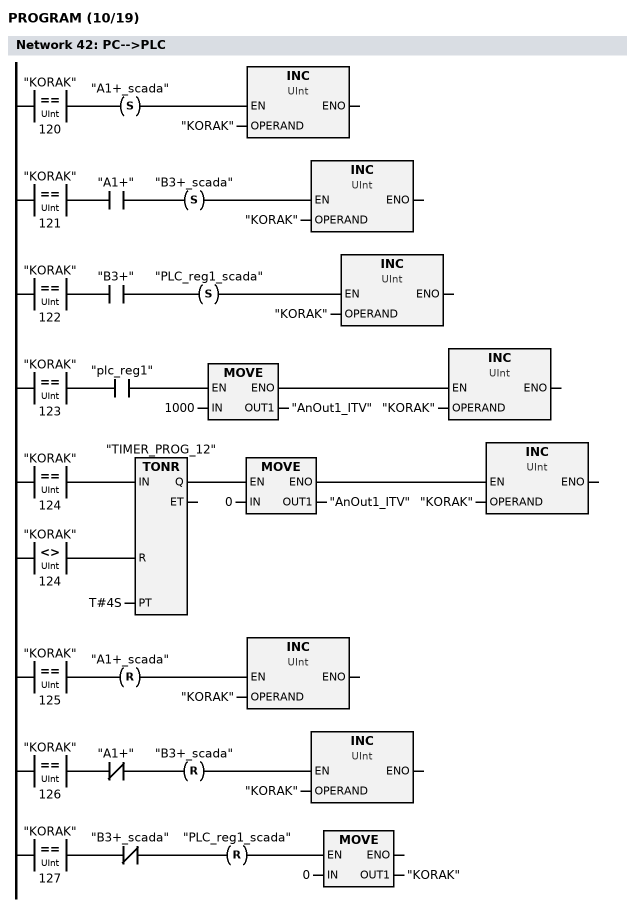
   IF "KORAK" = 120 THEN
       "A1+_scada" := TRUE;
       "KORAK" := "KORAK" + 1;
   END_IF;
   IF ("KORAK" = 121) AND "A1+" THEN
       "B3+_scada" := TRUE;
       "KORAK" := "KORAK" + 1;
   END_IF;
   IF ("KORAK" = 122) AND "B3+" THEN
       "PLC_reg1_scada" := TRUE;
       "KORAK" := "KORAK" + 1;
   END_IF;
   IF ("KORAK" = 123) AND "plc_reg1" THEN
       "AnOut1_ITV" := 1000;
       "KORAK" := "KORAK" + 1;
   END_IF;
   "TIMER_PROG_12".TONR(IN := "KORAK" = 124, R := "KORAK" <> 124, PT := T#4S);
   IF "TIMER_PROG_12".Q THEN
       "AnOut1_ITV" := 0;
       "KORAK" := "KORAK" + 1;
   END_IF;
   IF "KORAK" = 125 THEN
       "A1+_scada" := FALSE;
       "KORAK" := "KORAK" + 1;
   END_IF;
   IF ("KORAK" = 126) AND NOT "A1+" THEN
       "B3+_scada" := FALSE;
       "KORAK" := "KORAK" + 1;
   END_IF;
   IF ("KORAK" = 127) AND NOT "B3+_scada" THEN
       "PLC_reg1_scada" := FALSE;
       "KORAK" := 0;
   END_IF;
END_REGION

REGION Network 43: PC-->PLC
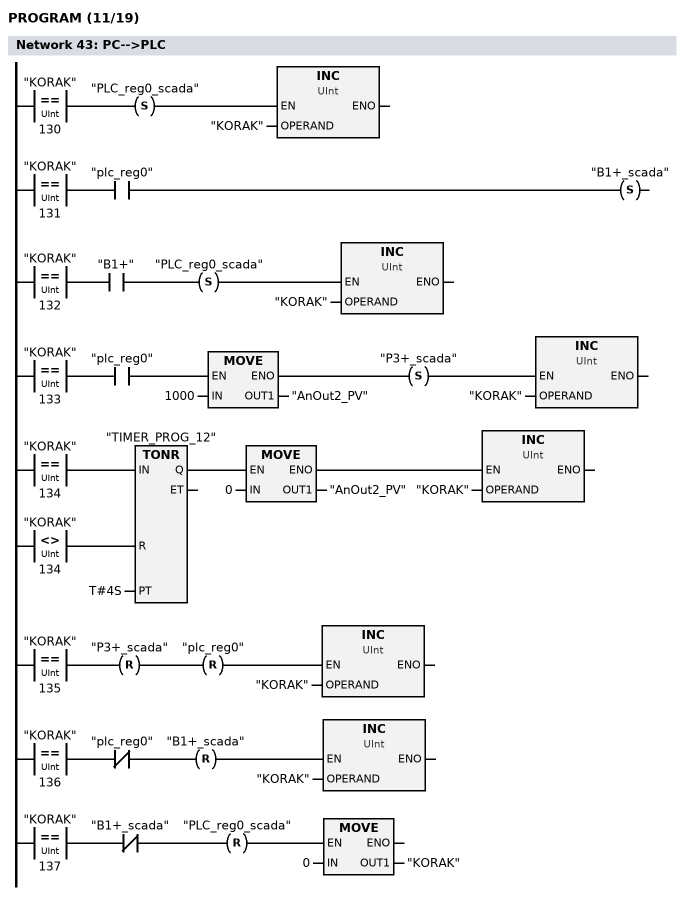
   IF "KORAK" = 130 THEN
       "PLC_reg0_scada" := TRUE;
       "KORAK" := "KORAK" + 1;
   END_IF;
   IF ("KORAK" = 131) AND "plc_reg0" THEN "B1+_scada" := TRUE; END_IF;
   IF ("KORAK" = 132) AND "B1+" THEN
       "PLC_reg0_scada" := TRUE;
       "KORAK" := "KORAK" + 1;
   END_IF;
   IF ("KORAK" = 133) AND "plc_reg0" THEN
       "AnOut2_PV" := 1000;
       "P3+_scada" := TRUE;
       "KORAK" := "KORAK" + 1;
   END_IF;
   "TIMER_PROG_12".TONR(IN := "KORAK" = 134, R := "KORAK" <> 134, PT := T#4S);
   IF "TIMER_PROG_12".Q THEN
       "AnOut2_PV" := 0;
       "KORAK" := "KORAK" + 1;
   END_IF;
   IF "KORAK" = 135 THEN
       "P3+_scada" := FALSE;
       "plc_reg0" := FALSE;
       "KORAK" := "KORAK" + 1;
   END_IF;
   IF ("KORAK" = 136) AND NOT "plc_reg0" THEN
       "B1+_scada" := FALSE;
       "KORAK" := "KORAK" + 1;
   END_IF;
   IF ("KORAK" = 137) AND NOT "B1+_scada" THEN
       "PLC_reg0_scada" := FALSE;
       "KORAK" := 0;
   END_IF;
END_REGION

REGION Network 44: PC-->PLC
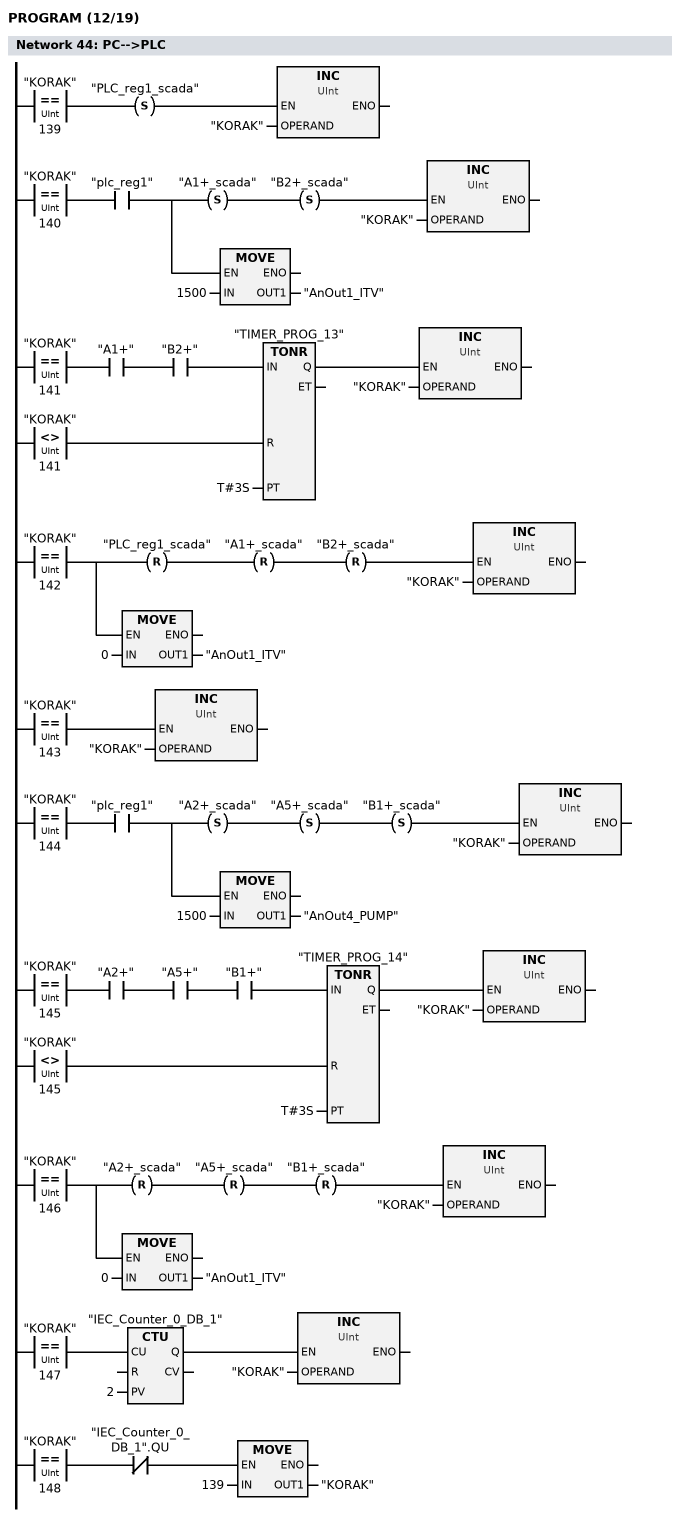
   IF "KORAK" = 139 THEN
       "PLC_reg1_scada" := TRUE;
       "KORAK" := "KORAK" + 1;
   END_IF;
   IF ("KORAK" = 140) AND "plc_reg1" THEN
       "A1+_scada" := TRUE;
       "B2+_scada" := TRUE;
   END_IF;
   #_w1 := ("KORAK" = 140) AND "plc_reg1";
   IF #_w1 THEN
       "KORAK" := "KORAK" + 1;
       "AnOut1_ITV" := 1500;
   END_IF;
   "TIMER_PROG_13".TONR(IN := ("KORAK" = 141) AND "A1+" AND "B2+", R := "KORAK" <> 141, PT := T#3S);
   IF "TIMER_PROG_13".Q THEN "KORAK" := "KORAK" + 1; END_IF;
   IF "KORAK" = 142 THEN
       "PLC_reg1_scada" := FALSE;
       "A1+_scada" := FALSE;
       "B2+_scada" := FALSE;
   END_IF;
   #_w2 := "KORAK" = 142;
   IF #_w2 THEN
       "KORAK" := "KORAK" + 1;
       "AnOut1_ITV" := 0;
   END_IF;
   IF "KORAK" = 143 THEN "KORAK" := "KORAK" + 1; END_IF;
   IF ("KORAK" = 144) AND "plc_reg1" THEN
       "A2+_scada" := TRUE;
       "A5+_scada" := TRUE;
       "B1+_scada" := TRUE;
   END_IF;
   #_w3 := ("KORAK" = 144) AND "plc_reg1";
   IF #_w3 THEN
       "KORAK" := "KORAK" + 1;
       "AnOut4_PUMP" := 1500;
   END_IF;
   "TIMER_PROG_14".TONR(IN := ("KORAK" = 145) AND "A2+" AND "A5+" AND "B1+", R := "KORAK" <> 145, PT := T#3S);
   IF "TIMER_PROG_14".Q THEN "KORAK" := "KORAK" + 1; END_IF;
   IF "KORAK" = 146 THEN
       "A2+_scada" := FALSE;
       "A5+_scada" := FALSE;
       "B1+_scada" := FALSE;
   END_IF;
   #_w4 := "KORAK" = 146;
   IF #_w4 THEN
       "KORAK" := "KORAK" + 1;
       "AnOut1_ITV" := 0;
   END_IF;
   "IEC_Counter_0_DB_1".CTU(CU := "KORAK" = 147, PV := 2);
   IF "IEC_Counter_0_DB_1".Q THEN "KORAK" := "KORAK" + 1; END_IF;
   IF ("KORAK" = 148) AND NOT "IEC_Counter_0_DB_1".QU THEN "KORAK" := 139; END_IF;
END_REGION

REGION Network 45: 2024_prva grupa
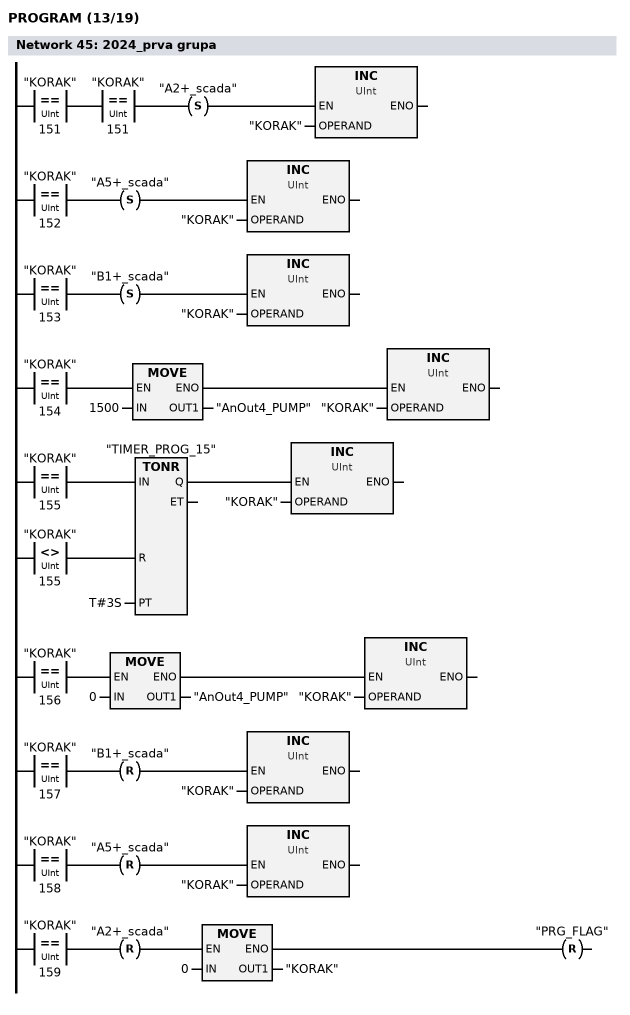
   IF ("KORAK" = 151) AND ("KORAK" = 151) THEN
       "A2+_scada" := TRUE;
       "KORAK" := "KORAK" + 1;
   END_IF;
   IF "KORAK" = 152 THEN
       "A5+_scada" := TRUE;
       "KORAK" := "KORAK" + 1;
   END_IF;
   IF "KORAK" = 153 THEN
       "B1+_scada" := TRUE;
       "KORAK" := "KORAK" + 1;
   END_IF;
   IF "KORAK" = 154 THEN
       "AnOut4_PUMP" := 1500;
       "KORAK" := "KORAK" + 1;
   END_IF;
   "TIMER_PROG_15".TONR(IN := "KORAK" = 155, R := "KORAK" <> 155, PT := T#3S);
   IF "TIMER_PROG_15".Q THEN "KORAK" := "KORAK" + 1; END_IF;
   IF "KORAK" = 156 THEN
       "AnOut4_PUMP" := 0;
       "KORAK" := "KORAK" + 1;
   END_IF;
   IF "KORAK" = 157 THEN
       "B1+_scada" := FALSE;
       "KORAK" := "KORAK" + 1;
   END_IF;
   IF "KORAK" = 158 THEN
       "A5+_scada" := FALSE;
       "KORAK" := "KORAK" + 1;
   END_IF;
   IF "KORAK" = 159 THEN "A2+_scada" := FALSE; END_IF;
   #_w1 := "KORAK" = 159;
   IF #_w1 THEN
       "KORAK" := 0;
       "PRG_FLAG" := FALSE;
   END_IF;
END_REGION

REGION Network 46: PC-->PLC
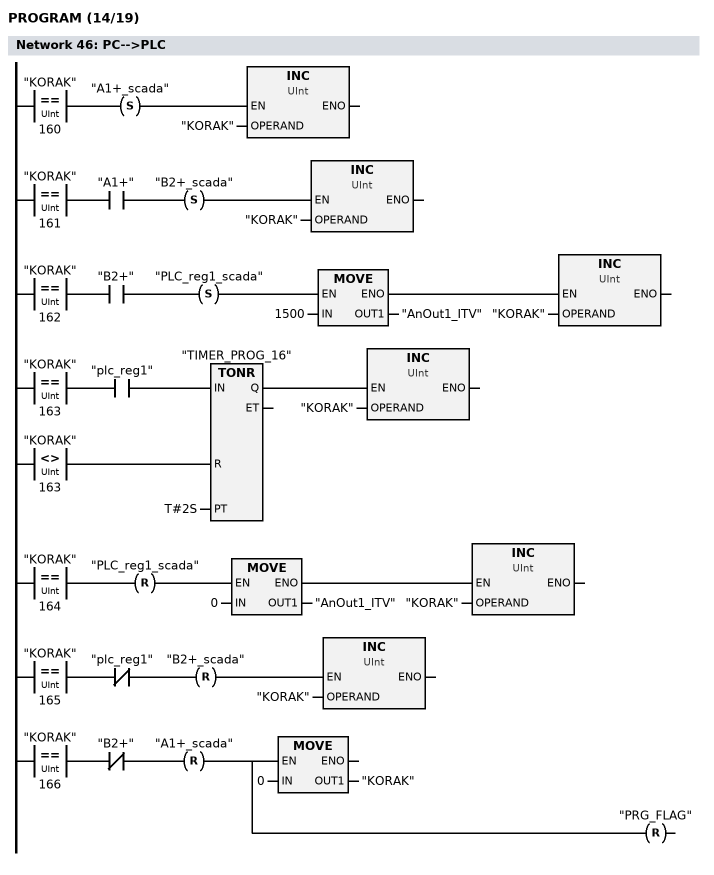
   IF "KORAK" = 160 THEN
       "A1+_scada" := TRUE;
       "KORAK" := "KORAK" + 1;
   END_IF;
   IF ("KORAK" = 161) AND "A1+" THEN
       "B2+_scada" := TRUE;
       "KORAK" := "KORAK" + 1;
   END_IF;
   IF ("KORAK" = 162) AND "B2+" THEN
       "PLC_reg1_scada" := TRUE;
       "AnOut1_ITV" := 1500;
       "KORAK" := "KORAK" + 1;
   END_IF;
   "TIMER_PROG_16".TONR(IN := ("KORAK" = 163) AND "plc_reg1", R := "KORAK" <> 163, PT := T#2S);
   IF "TIMER_PROG_16".Q THEN "KORAK" := "KORAK" + 1; END_IF;
   IF "KORAK" = 164 THEN
       "PLC_reg1_scada" := FALSE;
       "AnOut1_ITV" := 0;
       "KORAK" := "KORAK" + 1;
   END_IF;
   IF ("KORAK" = 165) AND NOT "plc_reg1" THEN
       "B2+_scada" := FALSE;
       "KORAK" := "KORAK" + 1;
   END_IF;
   IF ("KORAK" = 166) AND NOT "B2+" THEN "A1+_scada" := FALSE; END_IF;
   #_w1 := ("KORAK" = 166) AND NOT "B2+";
   IF #_w1 THEN
       "KORAK" := 0;
       "PRG_FLAG" := FALSE;
   END_IF;
END_REGION

REGION Network 47: PC-->PLC
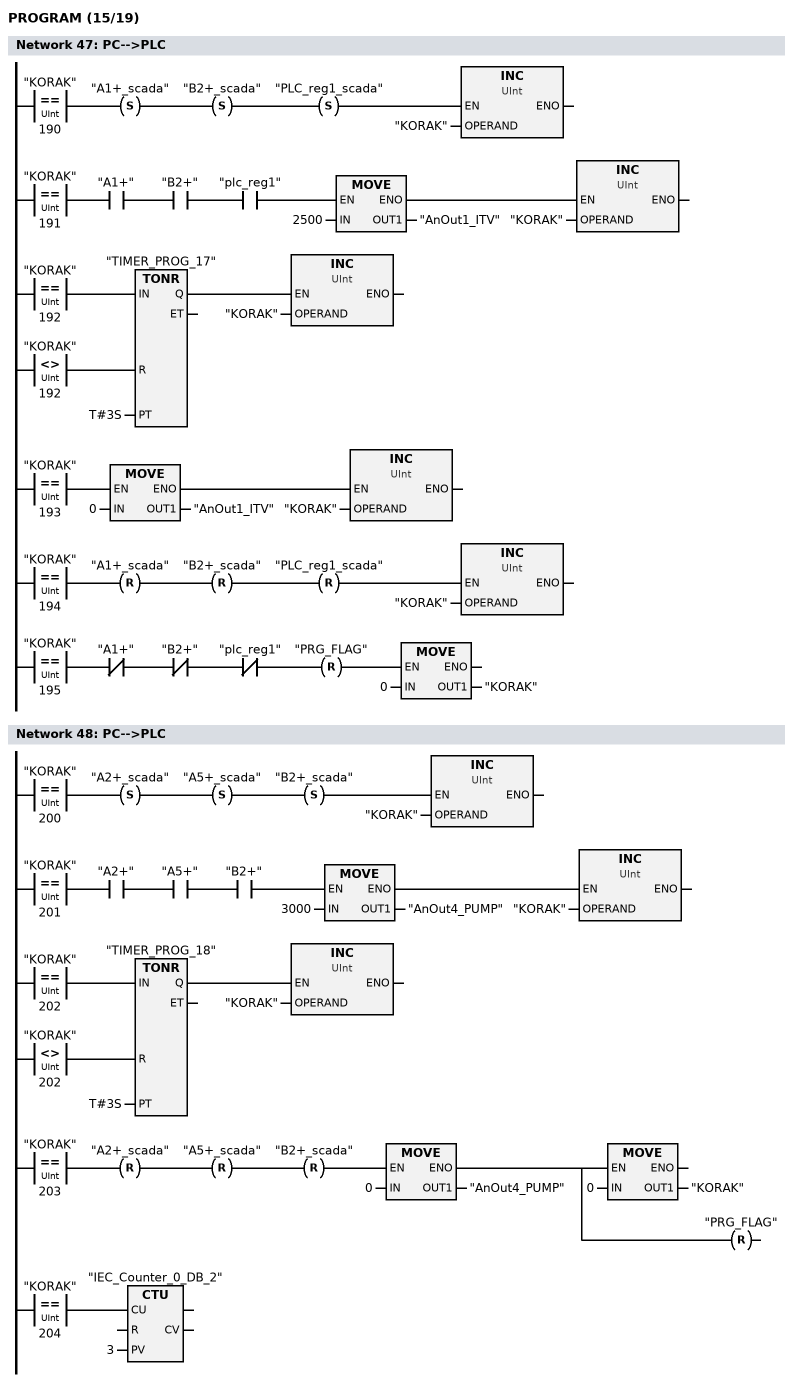
   IF "KORAK" = 190 THEN
       "A1+_scada" := TRUE;
       "B2+_scada" := TRUE;
       "PLC_reg1_scada" := TRUE;
       "KORAK" := "KORAK" + 1;
   END_IF;
   IF ("KORAK" = 191) AND "A1+" AND "B2+" AND "plc_reg1" THEN
       "AnOut1_ITV" := 2500;
       "KORAK" := "KORAK" + 1;
   END_IF;
   "TIMER_PROG_17".TONR(IN := "KORAK" = 192, R := "KORAK" <> 192, PT := T#3S);
   IF "TIMER_PROG_17".Q THEN "KORAK" := "KORAK" + 1; END_IF;
   IF "KORAK" = 193 THEN
       "AnOut1_ITV" := 0;
       "KORAK" := "KORAK" + 1;
   END_IF;
   IF "KORAK" = 194 THEN
       "A1+_scada" := FALSE;
       "B2+_scada" := FALSE;
       "PLC_reg1_scada" := FALSE;
       "KORAK" := "KORAK" + 1;
   END_IF;
   IF ("KORAK" = 195) AND NOT "A1+" AND NOT "B2+" AND NOT "plc_reg1" THEN
       "PRG_FLAG" := FALSE;
       "KORAK" := 0;
   END_IF;
END_REGION

REGION Network 48: PC-->PLC
   IF "KORAK" = 200 THEN
       "A2+_scada" := TRUE;
       "A5+_scada" := TRUE;
       "B2+_scada" := TRUE;
       "KORAK" := "KORAK" + 1;
   END_IF;
   IF ("KORAK" = 201) AND "A2+" AND "A5+" AND "B2+" THEN
       "AnOut4_PUMP" := 3000;
       "KORAK" := "KORAK" + 1;
   END_IF;
   "TIMER_PROG_18".TONR(IN := "KORAK" = 202, R := "KORAK" <> 202, PT := T#3S);
   IF "TIMER_PROG_18".Q THEN "KORAK" := "KORAK" + 1; END_IF;
   IF "KORAK" = 203 THEN
       "A2+_scada" := FALSE;
       "A5+_scada" := FALSE;
       "B2+_scada" := FALSE;
       "AnOut4_PUMP" := 0;
   END_IF;
   #_w1 := "KORAK" = 203;
   IF #_w1 THEN
       "KORAK" := 0;
       "PRG_FLAG" := FALSE;
   END_IF;
   "IEC_Counter_0_DB_2".CTU(CU := "KORAK" = 204, PV := 3);
END_REGION

REGION Network 49: PC-->PLC
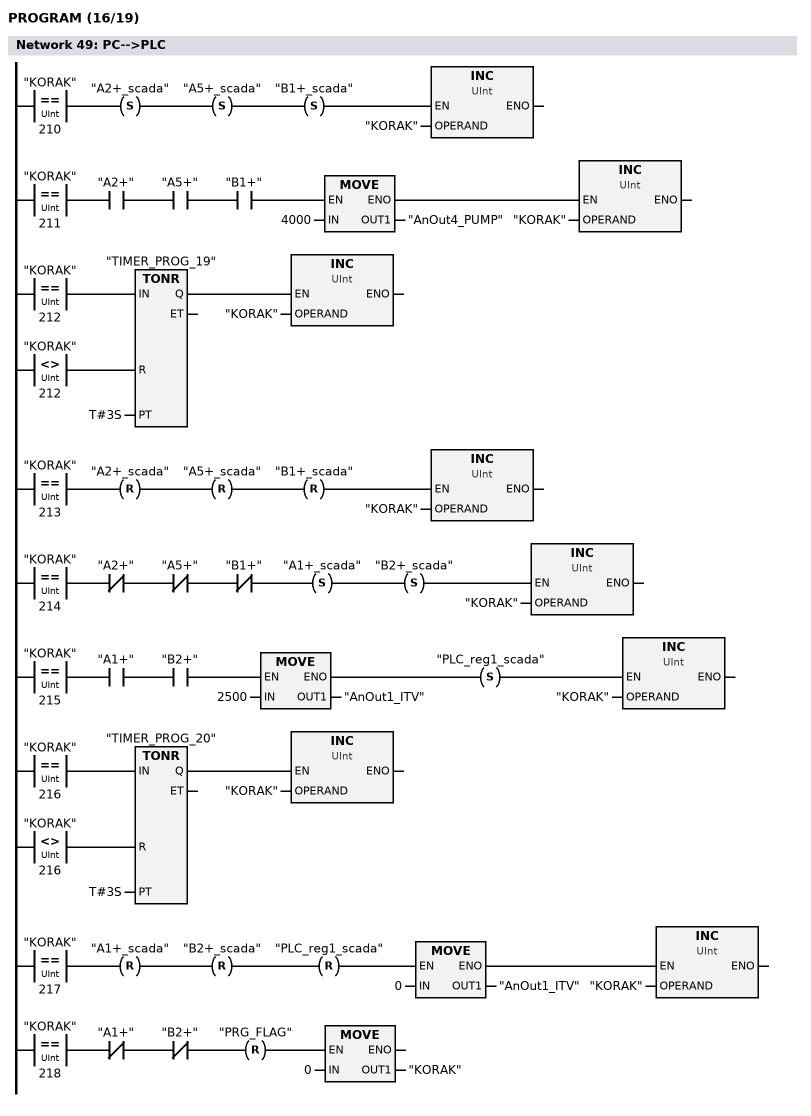
   IF "KORAK" = 210 THEN
       "A2+_scada" := TRUE;
       "A5+_scada" := TRUE;
       "B1+_scada" := TRUE;
       "KORAK" := "KORAK" + 1;
   END_IF;
   IF ("KORAK" = 211) AND "A2+" AND "A5+" AND "B1+" THEN
       "AnOut4_PUMP" := 4000;
       "KORAK" := "KORAK" + 1;
   END_IF;
   "TIMER_PROG_19".TONR(IN := "KORAK" = 212, R := "KORAK" <> 212, PT := T#3S);
   IF "TIMER_PROG_19".Q THEN "KORAK" := "KORAK" + 1; END_IF;
   IF "KORAK" = 213 THEN
       "A2+_scada" := FALSE;
       "A5+_scada" := FALSE;
       "B1+_scada" := FALSE;
       "KORAK" := "KORAK" + 1;
   END_IF;
   IF ("KORAK" = 214) AND NOT "A2+" AND NOT "A5+" AND NOT "B1+" THEN
       "A1+_scada" := TRUE;
       "B2+_scada" := TRUE;
       "KORAK" := "KORAK" + 1;
   END_IF;
   IF ("KORAK" = 215) AND "A1+" AND "B2+" THEN
       "AnOut1_ITV" := 2500;
       "PLC_reg1_scada" := TRUE;
       "KORAK" := "KORAK" + 1;
   END_IF;
   "TIMER_PROG_20".TONR(IN := "KORAK" = 216, R := "KORAK" <> 216, PT := T#3S);
   IF "TIMER_PROG_20".Q THEN "KORAK" := "KORAK" + 1; END_IF;
   IF "KORAK" = 217 THEN
       "A1+_scada" := FALSE;
       "B2+_scada" := FALSE;
       "PLC_reg1_scada" := FALSE;
       "AnOut1_ITV" := 0;
       "KORAK" := "KORAK" + 1;
   END_IF;
   IF ("KORAK" = 218) AND NOT "A1+" AND NOT "B2+" THEN
       "PRG_FLAG" := FALSE;
       "KORAK" := 0;
   END_IF;
END_REGION

REGION Network 50: PC-->PLC
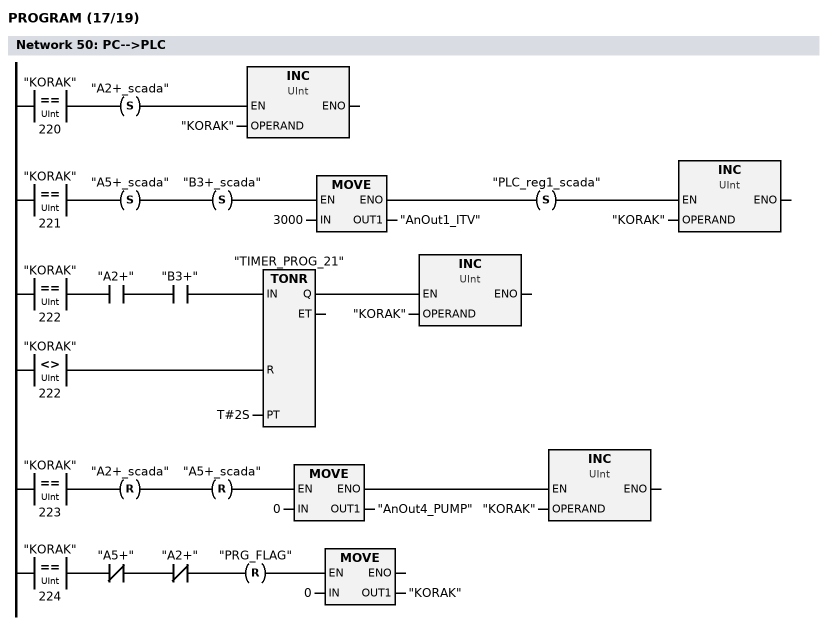
   IF "KORAK" = 220 THEN
       "A2+_scada" := TRUE;
       "KORAK" := "KORAK" + 1;
   END_IF;
   IF "KORAK" = 221 THEN
       "A5+_scada" := TRUE;
       "B3+_scada" := TRUE;
       "AnOut1_ITV" := 3000;
       "PLC_reg1_scada" := TRUE;
       "KORAK" := "KORAK" + 1;
   END_IF;
   "TIMER_PROG_21".TONR(IN := ("KORAK" = 222) AND "A2+" AND "B3+", R := "KORAK" <> 222, PT := T#2S);
   IF "TIMER_PROG_21".Q THEN "KORAK" := "KORAK" + 1; END_IF;
   IF "KORAK" = 223 THEN
       "A2+_scada" := FALSE;
       "A5+_scada" := FALSE;
       "AnOut4_PUMP" := 0;
       "KORAK" := "KORAK" + 1;
   END_IF;
   IF ("KORAK" = 224) AND NOT "A5+" AND NOT "A2+" THEN
       "PRG_FLAG" := FALSE;
       "KORAK" := 0;
   END_IF;
END_REGION

REGION Network 51: PC-->PLC
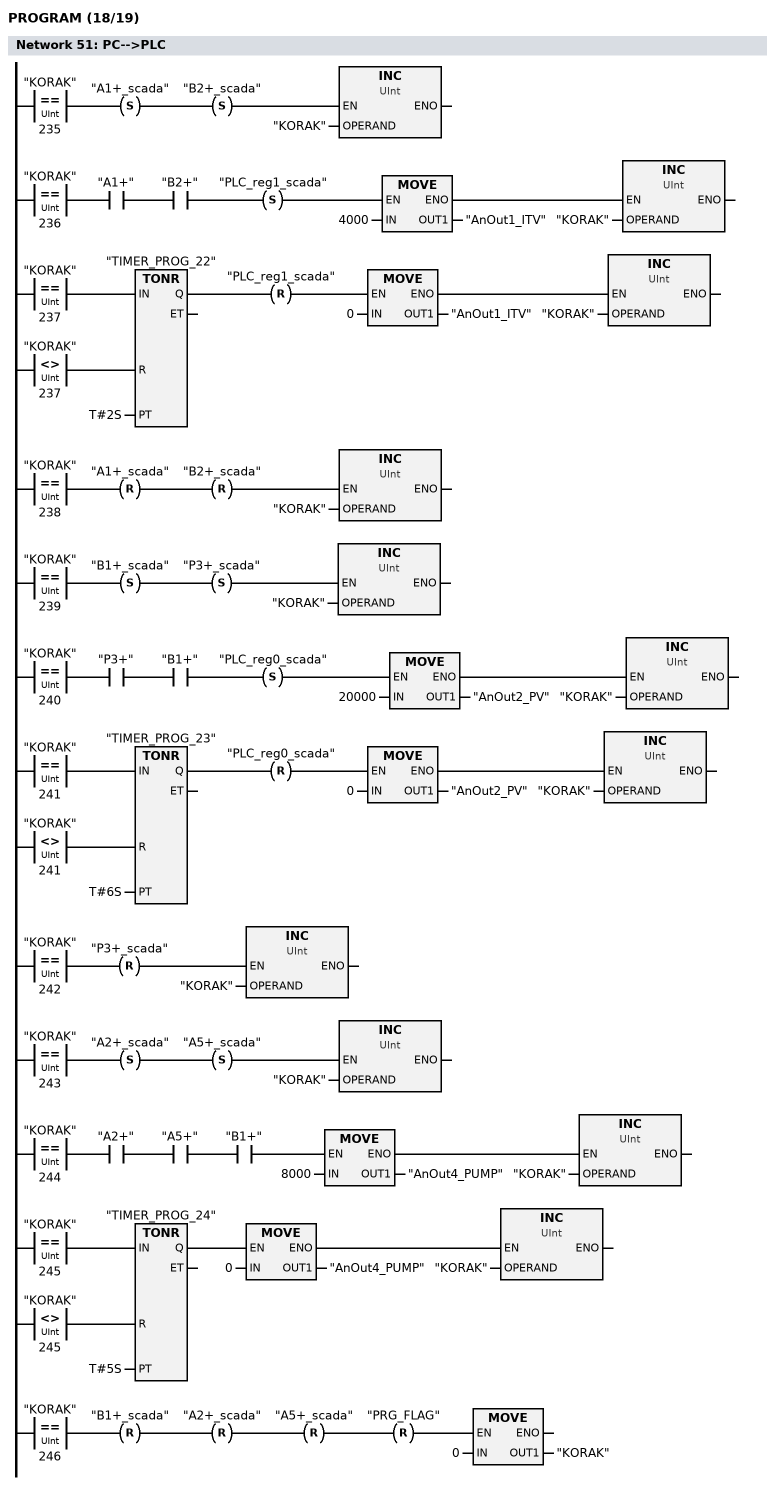
   IF "KORAK" = 235 THEN
       "A1+_scada" := TRUE;
       "B2+_scada" := TRUE;
       "KORAK" := "KORAK" + 1;
   END_IF;
   IF ("KORAK" = 236) AND "A1+" AND "B2+" THEN
       "PLC_reg1_scada" := TRUE;
       "AnOut1_ITV" := 4000;
       "KORAK" := "KORAK" + 1;
   END_IF;
   "TIMER_PROG_22".TONR(IN := "KORAK" = 237, R := "KORAK" <> 237, PT := T#2S);
   IF "TIMER_PROG_22".Q THEN
       "PLC_reg1_scada" := FALSE;
       "AnOut1_ITV" := 0;
       "KORAK" := "KORAK" + 1;
   END_IF;
   IF "KORAK" = 238 THEN
       "A1+_scada" := FALSE;
       "B2+_scada" := FALSE;
       "KORAK" := "KORAK" + 1;
   END_IF;
   IF "KORAK" = 239 THEN
       "B1+_scada" := TRUE;
       "P3+_scada" := TRUE;
       "KORAK" := "KORAK" + 1;
   END_IF;
   IF ("KORAK" = 240) AND "P3+" AND "B1+" THEN
       "PLC_reg0_scada" := TRUE;
       "AnOut2_PV" := 20000;
       "KORAK" := "KORAK" + 1;
   END_IF;
   "TIMER_PROG_23".TONR(IN := "KORAK" = 241, R := "KORAK" <> 241, PT := T#6S);
   IF "TIMER_PROG_23".Q THEN
       "PLC_reg0_scada" := FALSE;
       "AnOut2_PV" := 0;
       "KORAK" := "KORAK" + 1;
   END_IF;
   IF "KORAK" = 242 THEN
       "P3+_scada" := FALSE;
       "KORAK" := "KORAK" + 1;
   END_IF;
   IF "KORAK" = 243 THEN
       "A2+_scada" := TRUE;
       "A5+_scada" := TRUE;
       "KORAK" := "KORAK" + 1;
   END_IF;
   IF ("KORAK" = 244) AND "A2+" AND "A5+" AND "B1+" THEN
       "AnOut4_PUMP" := 8000;
       "KORAK" := "KORAK" + 1;
   END_IF;
   "TIMER_PROG_24".TONR(IN := "KORAK" = 245, R := "KORAK" <> 245, PT := T#5S);
   IF "TIMER_PROG_24".Q THEN
       "AnOut4_PUMP" := 0;
       "KORAK" := "KORAK" + 1;
   END_IF;
   IF "KORAK" = 246 THEN
       "B1+_scada" := FALSE;
       "A2+_scada" := FALSE;
       "A5+_scada" := FALSE;
       "PRG_FLAG" := FALSE;
       "KORAK" := 0;
   END_IF;
END_REGION

REGION Network 52: PC-->PLC
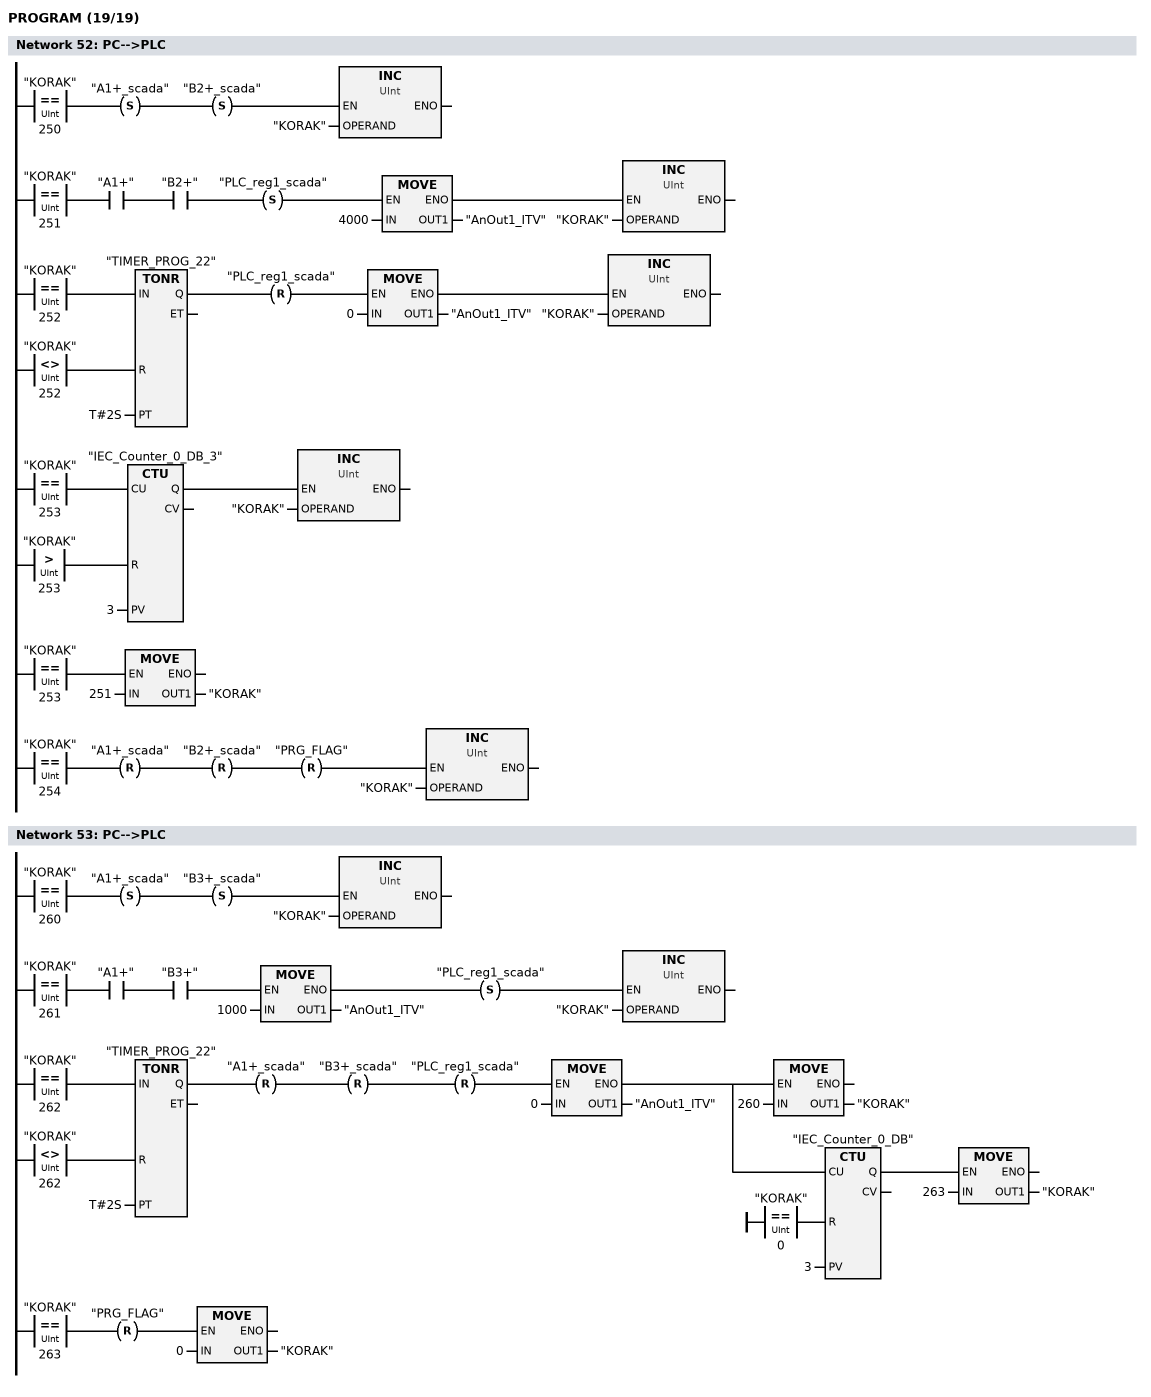
   IF "KORAK" = 250 THEN
       "A1+_scada" := TRUE;
       "B2+_scada" := TRUE;
       "KORAK" := "KORAK" + 1;
   END_IF;
   IF ("KORAK" = 251) AND "A1+" AND "B2+" THEN
       "PLC_reg1_scada" := TRUE;
       "AnOut1_ITV" := 4000;
       "KORAK" := "KORAK" + 1;
   END_IF;
   "TIMER_PROG_22".TONR(IN := "KORAK" = 252, R := "KORAK" <> 252, PT := T#2S);
   IF "TIMER_PROG_22".Q THEN
       "PLC_reg1_scada" := FALSE;
       "AnOut1_ITV" := 0;
       "KORAK" := "KORAK" + 1;
   END_IF;
   "IEC_Counter_0_DB_3".CTU(CU := "KORAK" = 253, R := "KORAK" > 253, PV := 3);
   IF "IEC_Counter_0_DB_3".Q THEN "KORAK" := "KORAK" + 1; END_IF;
   IF "KORAK" = 253 THEN "KORAK" := 251; END_IF;
   IF "KORAK" = 254 THEN
       "A1+_scada" := FALSE;
       "B2+_scada" := FALSE;
       "PRG_FLAG" := FALSE;
       "KORAK" := "KORAK" + 1;
   END_IF;
END_REGION

REGION Network 53: PC-->PLC
   IF "KORAK" = 260 THEN
       "A1+_scada" := TRUE;
       "B3+_scada" := TRUE;
       "KORAK" := "KORAK" + 1;
   END_IF;
   IF ("KORAK" = 261) AND "A1+" AND "B3+" THEN
       "AnOut1_ITV" := 1000;
       "PLC_reg1_scada" := TRUE;
       "KORAK" := "KORAK" + 1;
   END_IF;
   "TIMER_PROG_22".TONR(IN := "KORAK" = 262, R := "KORAK" <> 262, PT := T#2S);
   IF "TIMER_PROG_22".Q THEN
       "A1+_scada" := FALSE;
       "B3+_scada" := FALSE;
       "PLC_reg1_scada" := FALSE;
       "AnOut1_ITV" := 0;
       "KORAK" := 260;
   END_IF;
   "IEC_Counter_0_DB".CTU(CU := "TIMER_PROG_22".Q, R := "KORAK" = 0, PV := 3);
   IF "IEC_Counter_0_DB".Q THEN "KORAK" := 263; END_IF;
   IF "KORAK" = 263 THEN
       "PRG_FLAG" := FALSE;
       "KORAK" := 0;
   END_IF;
END_REGION
END_FUNCTION

FUNCTION "STOP_LOAD_TANK" : Void   // FC8, SCL
{ S7_Optimized_Access := 'TRUE' }
VERSION : 0.1
   VAR_OUTPUT
      command1 : Bool;
      command2 : Bool;
      command3 : Bool;
      pumpOutput : Int;
   END_VAR
BEGIN
   #command1 := FALSE;
   #command2 := FALSE;
   #command3 := FALSE;
   #pumpOutput := 0;
END_FUNCTION

FUNCTION "START_LOAD_APPLE_JUICE_TANK" : Void   // FC9, SCL
{ S7_Optimized_Access := 'TRUE' }
VERSION : 0.1
   VAR_INPUT
      feedback1 : Bool;
      feedback2 : Bool;
      analogValue : Int;
   END_VAR
   VAR_OUTPUT
      command1 : Bool;
      command2 : Bool;
      regulatorCommand : Bool;
      analogOutput : Int;
      routeReady : Bool;
   END_VAR
BEGIN
   #command1 := TRUE;
   #command2 := TRUE;

   IF #feedback1 = TRUE AND #feedback2 = TRUE THEN
       #regulatorCommand := TRUE;
       #analogOutput := #analogValue;
       #routeReady := TRUE;
   ELSE
       #regulatorCommand := FALSE;
       #analogOutput := 0;
       #routeReady := FALSE;
   END_IF;
END_FUNCTION

FUNCTION "STOP_LOAD_APPLE_JUICE_TANK" : Void   // FC10, SCL
{ S7_Optimized_Access := 'TRUE' }
VERSION : 0.1
   VAR_OUTPUT
      command1 : Bool;
      command2 : Bool;
      regulatorCommand : Bool;
      analogOutput : Int;
   END_VAR
BEGIN
   #command1 := FALSE;
   #command2 := FALSE;
   #regulatorCommand := FALSE;
   #analogOutput := 0;
END_FUNCTION

FUNCTION "START_LOAD_TANK" : Void   // FC11, SCL
{ S7_Optimized_Access := 'TRUE' }
VERSION : 0.1
   VAR_INPUT
      feedback1 : Bool;
      feedback2 : Bool;
      feedback3 : Bool;
      pumpValue : Int;
   END_VAR
   VAR_OUTPUT
      command1 : Bool;
      command2 : Bool;
      command3 : Bool;
      pumpOutput : Int;
      routeReady : Bool;
   END_VAR
BEGIN
   #command1 := TRUE;
   #command2 := TRUE;
   #command3 := TRUE;

   IF #feedback1 = TRUE AND #feedback2 = TRUE AND #feedback3 = TRUE THEN
       #pumpOutput := #pumpValue;
       #routeReady := TRUE;
   ELSE
       #pumpOutput := 0;
       #routeReady := FALSE;
   END_IF;
END_FUNCTION

FUNCTION "FILL_APPLE_TO_BOTTLE" : Void   // FC12, SCL
{ S7_Optimized_Access := 'TRUE' }
VERSION : 0.1
   VAR_INPUT
      feedback1 : Bool;
      feedback2 : Bool;
      analogValue : Int;
   END_VAR
   VAR_OUTPUT
      command1 : Bool;
      command2 : Bool;
      analogOutput : Int;
      routeReady : Bool;
   END_VAR
BEGIN
   #command1 := TRUE;
   #command2 := TRUE;

   IF #feedback1 = TRUE AND #feedback2 = TRUE THEN
       #analogOutput := #analogValue;
       #routeReady := TRUE;
   ELSE;
       #analogOutput := 0;
       #routeReady := FALSE;
   END_IF;
END_FUNCTION

FUNCTION "STOP_FILL_APPLE_TO_BOTTLE" : Void   // FC13, SCL
{ S7_Optimized_Access := 'TRUE' }
VERSION : 0.1
   VAR_OUTPUT
      command1 : Bool;
      command2 : Bool;
      analogOutput : Int;
   END_VAR
BEGIN
   #command1 := FALSE;
   #command2 := FALSE;
   #analogOutput := 0;
END_FUNCTION

ORGANIZATION_BLOCK "Main"   // OB1, LAD, ProgramCycle
TITLE = "Main Program Sweep (Cycle)"
{ S7_Optimized_Access := 'TRUE' }
VERSION : 0.1
BEGIN

REGION Network 1: Analog pressure of the TANK 1
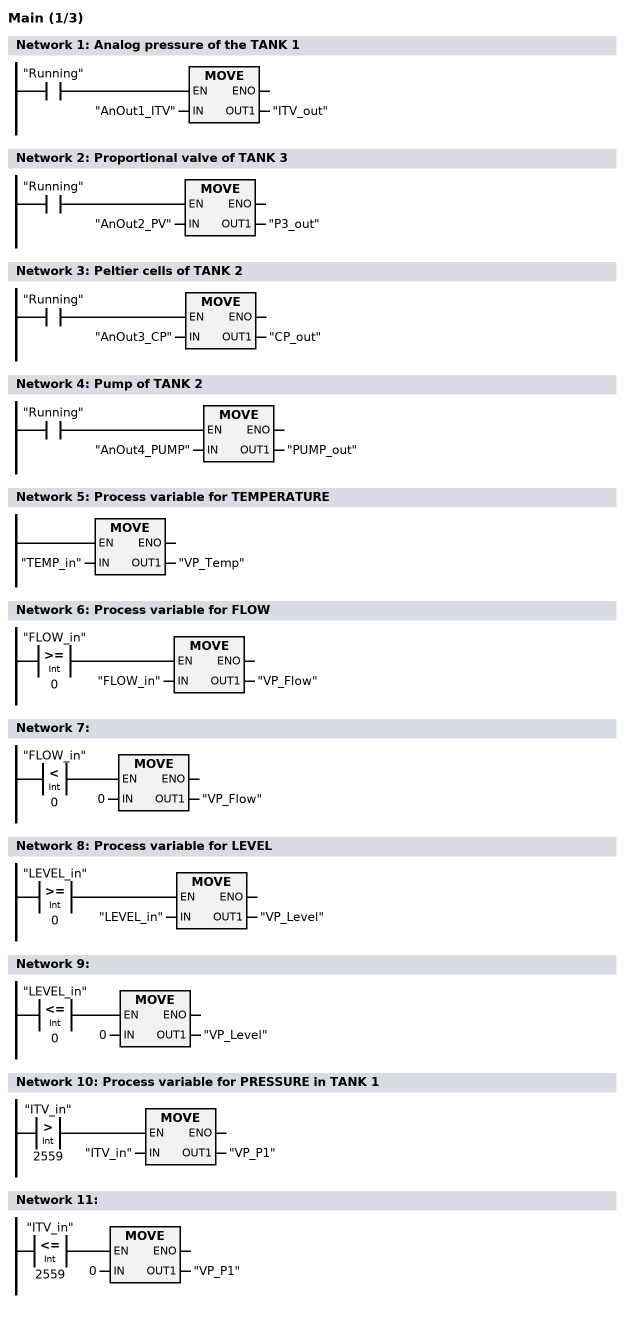
   RUNG wire#powerrail
      Contact( "Running" )
      { S7_GenerateENO := "TRUE" } Move(in := "AnOut1_ITV", out1 => "ITV_out")
   END_RUNG
   // the same network as SCL:
   IF "Running" THEN "ITV_out" := "AnOut1_ITV"; END_IF;
END_REGION

REGION Network 2: Proportional valve of TANK 3
   RUNG wire#powerrail
      Contact( "Running" )
      { S7_GenerateENO := "TRUE" } Move(in := "AnOut2_PV", out1 => "P3_out")
   END_RUNG
   // the same network as SCL:
   IF "Running" THEN "P3_out" := "AnOut2_PV"; END_IF;
END_REGION

REGION Network 3: Peltier cells of TANK 2
   RUNG wire#powerrail
      Contact( "Running" )
      { S7_GenerateENO := "TRUE" } Move(in := "AnOut3_CP", out1 => "CP_out")
   END_RUNG
   // the same network as SCL:
   IF "Running" THEN "CP_out" := "AnOut3_CP"; END_IF;
END_REGION

REGION Network 4: Pump of TANK 2
   RUNG wire#powerrail
      Contact( "Running" )
      { S7_GenerateENO := "TRUE" } Move(in := "AnOut4_PUMP", out1 => "PUMP_out")
   END_RUNG
   // the same network as SCL:
   IF "Running" THEN "PUMP_out" := "AnOut4_PUMP"; END_IF;
END_REGION

REGION Network 5: Process variable for TEMPERATURE
   RUNG wire#powerrail
      { S7_GenerateENO := "TRUE" } Move(in := "TEMP_in", out1 => "VP_Temp")
   END_RUNG
   // the same network as SCL:
   "VP_Temp" := "TEMP_in";
END_REGION

REGION Network 6: Process variable for FLOW
   RUNG wire#powerrail
      { S7_Templates := "SrcType := Int" } GE_Contact(in1 := "FLOW_in", in2 := 0)
      { S7_GenerateENO := "TRUE" } Move(in := "FLOW_in", out1 => "VP_Flow")
   END_RUNG
   // the same network as SCL:
   IF "FLOW_in" >= 0 THEN "VP_Flow" := "FLOW_in"; END_IF;
END_REGION

REGION Network 7
   RUNG wire#powerrail
      { S7_Templates := "SrcType := Int" } LT_Contact(in1 := "FLOW_in", in2 := 0)
      { S7_GenerateENO := "TRUE" } Move(in := 0, out1 => "VP_Flow")
   END_RUNG
   // the same network as SCL:
   IF "FLOW_in" < 0 THEN "VP_Flow" := 0; END_IF;
END_REGION

REGION Network 8: Process variable for LEVEL
   RUNG wire#powerrail
      { S7_Templates := "SrcType := Int" } GE_Contact(in1 := "LEVEL_in", in2 := 0)
      { S7_GenerateENO := "TRUE" } Move(in := "LEVEL_in", out1 => "VP_Level")
   END_RUNG
   // the same network as SCL:
   IF "LEVEL_in" >= 0 THEN "VP_Level" := "LEVEL_in"; END_IF;
END_REGION

REGION Network 9
   RUNG wire#powerrail
      { S7_Templates := "SrcType := Int" } LE_Contact(in1 := "LEVEL_in", in2 := 0)
      { S7_GenerateENO := "TRUE" } Move(in := 0, out1 => "VP_Level")
   END_RUNG
   // the same network as SCL:
   IF "LEVEL_in" <= 0 THEN "VP_Level" := 0; END_IF;
END_REGION

REGION Network 10: Process variable for PRESSURE in TANK 1
   RUNG wire#powerrail
      { S7_Templates := "SrcType := Int" } GT_Contact(in1 := "ITV_in", in2 := 2559)
      { S7_GenerateENO := "TRUE" } Move(in := "ITV_in", out1 => "VP_P1")
   END_RUNG
   // the same network as SCL:
   IF "ITV_in" > 2559 THEN "VP_P1" := "ITV_in"; END_IF;
END_REGION

REGION Network 11
   RUNG wire#powerrail
      { S7_Templates := "SrcType := Int" } LE_Contact(in1 := "ITV_in", in2 := 2559)
      { S7_GenerateENO := "TRUE" } Move(in := 0, out1 => "VP_P1")
   END_RUNG
   // the same network as SCL:
   IF "ITV_in" <= 2559 THEN "VP_P1" := 0; END_IF;
END_REGION

REGION Network 12: Process variable for PRESSURE in TANK 3
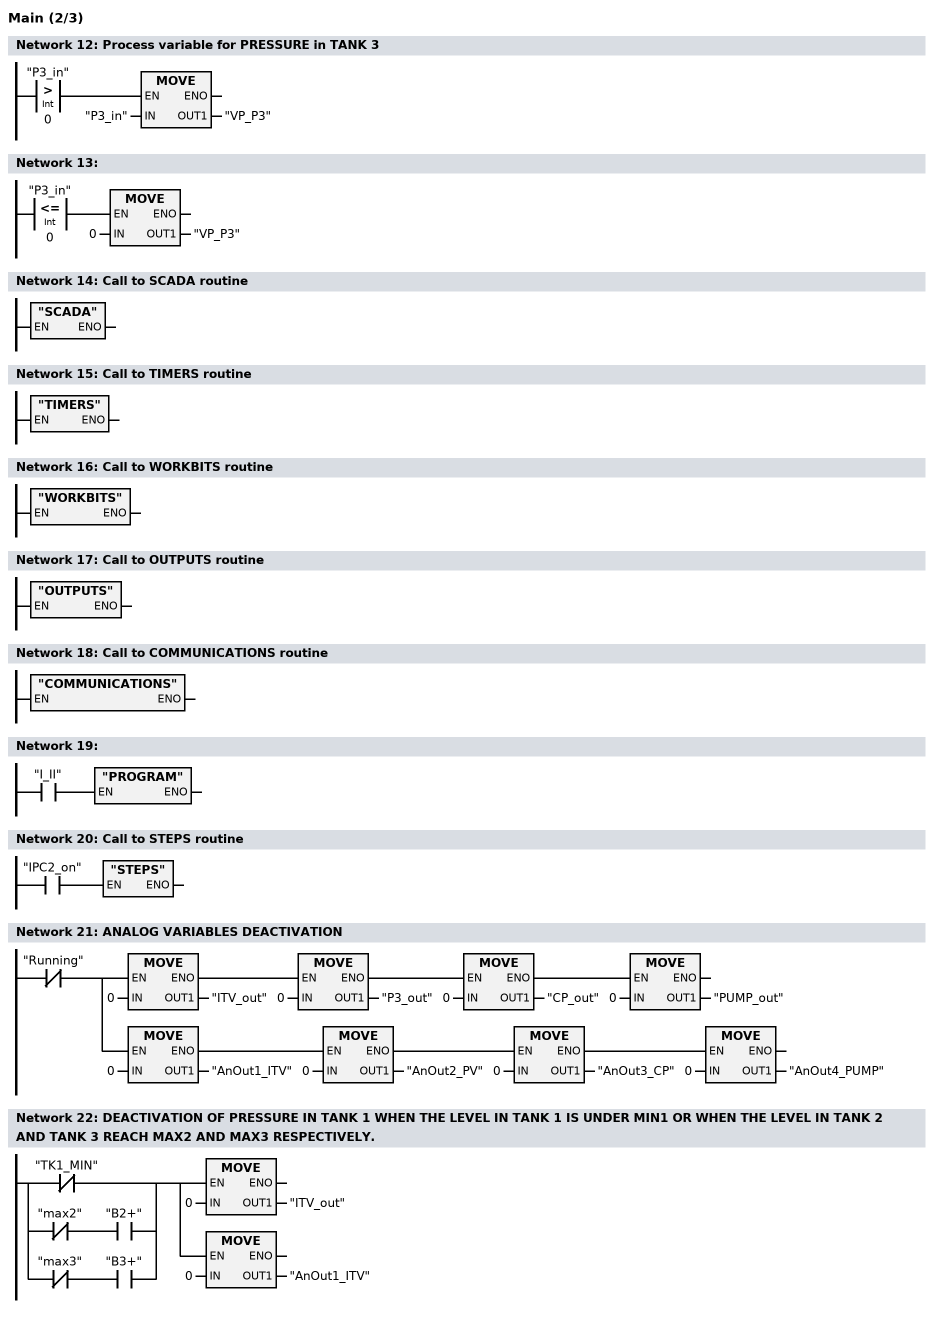
   RUNG wire#powerrail
      { S7_Templates := "SrcType := Int" } GT_Contact(in1 := "P3_in", in2 := 0)
      { S7_GenerateENO := "TRUE" } Move(in := "P3_in", out1 => "VP_P3")
   END_RUNG
   // the same network as SCL:
   IF "P3_in" > 0 THEN "VP_P3" := "P3_in"; END_IF;
END_REGION

REGION Network 13
   RUNG wire#powerrail
      { S7_Templates := "SrcType := Int" } LE_Contact(in1 := "P3_in", in2 := 0)
      { S7_GenerateENO := "TRUE" } Move(in := 0, out1 => "VP_P3")
   END_RUNG
   // the same network as SCL:
   IF "P3_in" <= 0 THEN "VP_P3" := 0; END_IF;
END_REGION

REGION Network 14: Call to SCADA routine
   RUNG wire#powerrail
      "SCADA"()
   END_RUNG
   // the same network as SCL:
   "SCADA"();
END_REGION

REGION Network 15: Call to TIMERS routine
   RUNG wire#powerrail
      "TIMERS"()
   END_RUNG
   // the same network as SCL:
   "TIMERS"();
END_REGION

REGION Network 16: Call to WORKBITS routine
   RUNG wire#powerrail
      "WORKBITS"()
   END_RUNG
   // the same network as SCL:
   "WORKBITS"();
END_REGION

REGION Network 17: Call to OUTPUTS routine
   RUNG wire#powerrail
      "OUTPUTS"()
   END_RUNG
   // the same network as SCL:
   "OUTPUTS"();
END_REGION

REGION Network 18: Call to COMMUNICATIONS routine
   RUNG wire#powerrail
      "COMMUNICATIONS"()
   END_RUNG
   // the same network as SCL:
   "COMMUNICATIONS"();
END_REGION

REGION Network 19
   RUNG wire#powerrail
      Contact( "I_II" )
      "PROGRAM"()
   END_RUNG
   // the same network as SCL:
   IF "I_II" THEN "PROGRAM"(); END_IF;
END_REGION

REGION Network 20: Call to STEPS routine
   RUNG wire#powerrail
      Contact( "IPC2_on" )
      "STEPS"()
   END_RUNG
   // the same network as SCL:
   IF "IPC2_on" THEN "STEPS"(); END_IF;
END_REGION

REGION Network 21: ANALOG VARIABLES DEACTIVATION
   RUNG wire#powerrail
      I_Contact( "Running" )
      wire#w1
      { S7_GenerateENO := "TRUE" } Move(in := 0, out1 => "ITV_out")
      { S7_GenerateENO := "TRUE" } Move(in := 0, out1 => "P3_out")
      { S7_GenerateENO := "TRUE" } Move(in := 0, out1 => "CP_out")
      { S7_GenerateENO := "TRUE" } Move(in := 0, out1 => "PUMP_out")
   END_RUNG
   RUNG wire#w1
      { S7_GenerateENO := "TRUE" } Move(in := 0, out1 => "AnOut1_ITV")
      { S7_GenerateENO := "TRUE" } Move(in := 0, out1 => "AnOut2_PV")
      { S7_GenerateENO := "TRUE" } Move(in := 0, out1 => "AnOut3_CP")
      { S7_GenerateENO := "TRUE" } Move(in := 0, out1 => "AnOut4_PUMP")
   END_RUNG
   // the same network as SCL:
   // ENO of a box is taken as its EN; it also drops when the box reports an error
   IF NOT "Running" THEN
       "ITV_out" := 0;
       "P3_out" := 0;
       "CP_out" := 0;
       "PUMP_out" := 0;
       "AnOut1_ITV" := 0;
       "AnOut2_PV" := 0;
       "AnOut3_CP" := 0;
       "AnOut4_PUMP" := 0;
   END_IF;
END_REGION

REGION Network 22: DEACTIVATION OF PRESSURE IN TANK 1 WHEN THE LEVEL IN TANK 1 IS UNDER MIN1 OR WHEN THE LEVEL IN TANK 2 AND TANK 3 REACH MAX2 AND MAX3 RESPECTIVELY.
   RUNG wire#powerrail
      I_Contact( "TK1_MIN" )
      wire#w1
      { S7_GenerateENO := "TRUE" } Move(in := 0, out1 => "ITV_out")
   END_RUNG
   RUNG wire#powerrail
      I_Contact( "max2" )
      Contact( "B2+" )
   END_RUNG wire#w1
   RUNG wire#powerrail
      I_Contact( "max3" )
      Contact( "B3+" )
   END_RUNG wire#w1
   RUNG wire#w1
      { S7_GenerateENO := "TRUE" } Move(in := 0, out1 => "AnOut1_ITV")
   END_RUNG
   // the same network as SCL:
   IF NOT "TK1_MIN" OR (NOT "max2" AND "B2+") OR (NOT "max3" AND "B3+") THEN
       "ITV_out" := 0;
       "AnOut1_ITV" := 0;
   END_IF;
END_REGION

REGION Network 23: DEACTIVATION OF THE PUMP WHEN THE LEVEL IN TANK 2 IS UNDER MIN2 OR WHEN THE LEVEL IN WHICHEVER TANK REACHES THE MAX LEVEL.
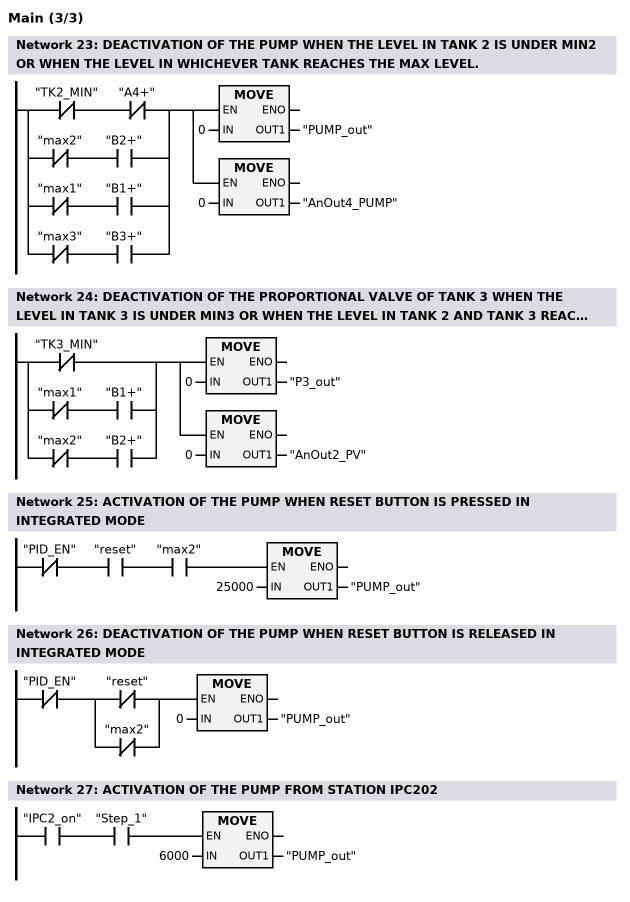
   RUNG wire#powerrail
      I_Contact( "TK2_MIN" )
      I_Contact( "A4+" )
      wire#w1
      { S7_GenerateENO := "TRUE" } Move(in := 0, out1 => "PUMP_out")
   END_RUNG
   RUNG wire#powerrail
      I_Contact( "max2" )
      Contact( "B2+" )
   END_RUNG wire#w1
   RUNG wire#powerrail
      I_Contact( "max1" )
      Contact( "B1+" )
   END_RUNG wire#w1
   RUNG wire#powerrail
      I_Contact( "max3" )
      Contact( "B3+" )
   END_RUNG wire#w1
   RUNG wire#w1
      { S7_GenerateENO := "TRUE" } Move(in := 0, out1 => "AnOut4_PUMP")
   END_RUNG
   // the same network as SCL:
   IF (NOT "TK2_MIN" AND NOT "A4+") OR (NOT "max2" AND "B2+") OR (NOT "max1" AND "B1+") OR (NOT "max3" AND "B3+") THEN
       "PUMP_out" := 0;
       "AnOut4_PUMP" := 0;
   END_IF;
END_REGION

REGION Network 24: DEACTIVATION OF THE PROPORTIONAL VALVE OF TANK 3 WHEN THE LEVEL IN TANK 3 IS UNDER MIN3 OR WHEN THE LEVEL IN TANK 2 AND TANK 3 REACH MAX2 AND MAX3 RESPECTIVELY
   RUNG wire#powerrail
      I_Contact( "TK3_MIN" )
      wire#w1
      { S7_GenerateENO := "TRUE" } Move(in := 0, out1 => "P3_out")
   END_RUNG
   RUNG wire#powerrail
      I_Contact( "max1" )
      Contact( "B1+" )
   END_RUNG wire#w1
   RUNG wire#powerrail
      I_Contact( "max2" )
      Contact( "B2+" )
   END_RUNG wire#w1
   RUNG wire#w1
      { S7_GenerateENO := "TRUE" } Move(in := 0, out1 => "AnOut2_PV")
   END_RUNG
   // the same network as SCL:
   IF NOT "TK3_MIN" OR (NOT "max1" AND "B1+") OR (NOT "max2" AND "B2+") THEN
       "P3_out" := 0;
       "AnOut2_PV" := 0;
   END_IF;
END_REGION

REGION Network 25: ACTIVATION OF THE PUMP WHEN RESET BUTTON IS PRESSED IN INTEGRATED MODE
   RUNG wire#powerrail
      I_Contact( "PID_EN" )
      Contact( "reset" )
      Contact( "max2" )
      { S7_GenerateENO := "TRUE" } Move(in := 25000, out1 => "PUMP_out")
   END_RUNG
   // the same network as SCL:
   IF NOT "PID_EN" AND "reset" AND "max2" THEN "PUMP_out" := 25000; END_IF;
END_REGION

REGION Network 26: DEACTIVATION OF THE PUMP WHEN RESET BUTTON IS RELEASED IN INTEGRATED MODE
   RUNG wire#powerrail
      I_Contact( "PID_EN" )
      wire#w1
      I_Contact( "reset" )
      wire#w2
      { S7_GenerateENO := "TRUE" } Move(in := 0, out1 => "PUMP_out")
   END_RUNG
   RUNG wire#w1
      I_Contact( "max2" )
   END_RUNG wire#w2
   // the same network as SCL:
   IF NOT "PID_EN" AND (NOT "reset" OR NOT "max2") THEN "PUMP_out" := 0; END_IF;
END_REGION

REGION Network 27: ACTIVATION OF THE PUMP FROM STATION IPC202
   RUNG wire#powerrail
      Contact( "IPC2_on" )
      Contact( "Step_1" )
      { S7_GenerateENO := "TRUE" } Move(in := 6000, out1 => "PUMP_out")
   END_RUNG
   // the same network as SCL:
   IF "IPC2_on" AND "Step_1" THEN "PUMP_out" := 6000; END_IF;
END_REGION
END_ORGANIZATION_BLOCK

ORGANIZATION_BLOCK "Startup"   // OB100, LAD, Startup
TITLE = "Complete Restart"
{ S7_Optimized_Access := 'TRUE' }
VERSION : 0.1
   VAR_INPUT
      LostRetentive : Bool;   // True if retentive data are lost
      LostRTC : Bool;   // True if date and time are lost
   END_VAR
BEGIN

REGION Network 1: SET the STEP 0 of the Grafcet
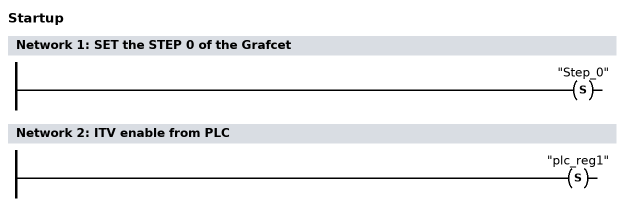
   RUNG wire#powerrail
      S_Coil( "Step_0" )
   END_RUNG
   // the same network as SCL:
   "Step_0" := TRUE;
END_REGION

REGION Network 2: ITV enable from PLC
   RUNG wire#powerrail
      S_Coil( "plc_reg1" )
   END_RUNG
   // the same network as SCL:
   "plc_reg1" := TRUE;
END_REGION
END_ORGANIZATION_BLOCK

ORGANIZATION_BLOCK "PID"   // OB200, LAD, CyclicInterrupt
TITLE = PID EXERCISES
{ S7_Optimized_Access := 'TRUE' }
VERSION : 0.1
BEGIN

REGION Network 1: CLOSED LOOP FOR THE TEMPERATURE EXERCISE (HEATING & COOLING)
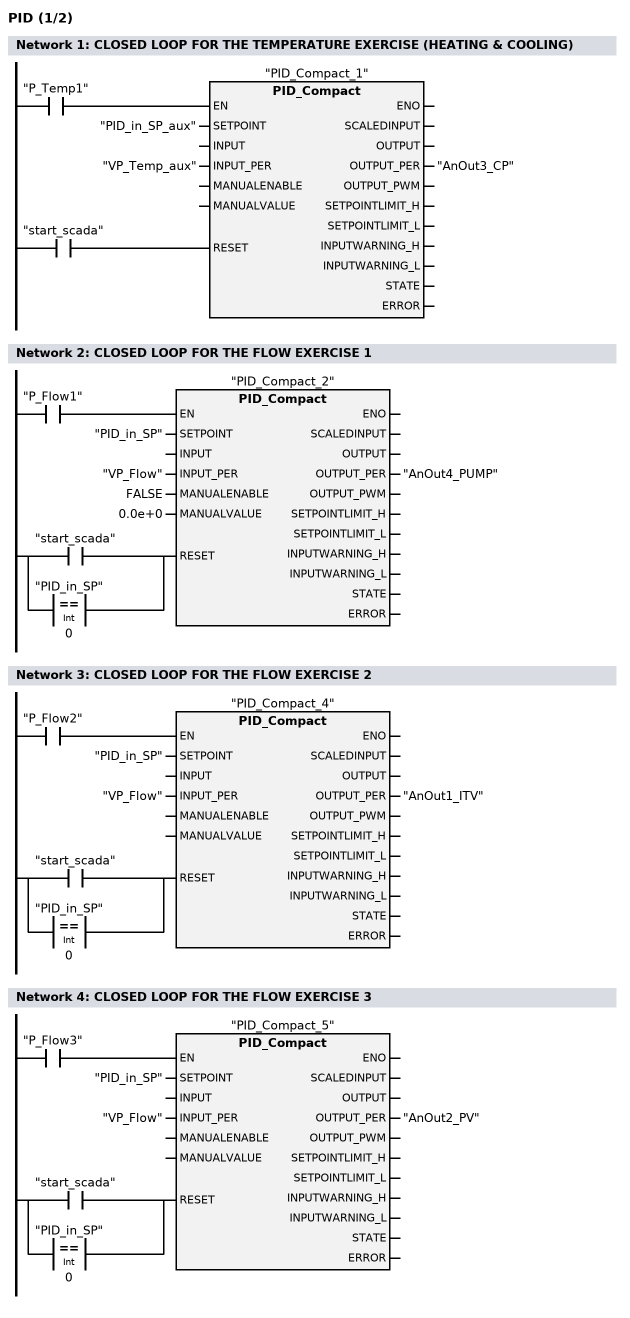
   IF "P_Temp1" THEN
       "PID_Compact_1"(Setpoint := "PID_in_SP_aux",   // PID_Compact
                       Input_PER := "VP_Temp_aux",
                       Reset := "start_scada",
                       Output_PER => "AnOut3_CP");
   END_IF;
END_REGION

REGION Network 2: CLOSED LOOP FOR THE FLOW EXERCISE 1
   IF "P_Flow1" THEN
       "PID_Compact_2"(Setpoint := "PID_in_SP",   // PID_Compact
                       Input_PER := "VP_Flow",
                       ManualEnable := FALSE,
                       ManualValue := 0.0e+0,
                       Reset := "start_scada" OR ("PID_in_SP" = 0),
                       Output_PER => "AnOut4_PUMP");
   END_IF;
END_REGION

REGION Network 3: CLOSED LOOP FOR THE FLOW EXERCISE 2
   IF "P_Flow2" THEN
       "PID_Compact_4"(Setpoint := "PID_in_SP",   // PID_Compact
                       Input_PER := "VP_Flow",
                       Reset := "start_scada" OR ("PID_in_SP" = 0),
                       Output_PER => "AnOut1_ITV");
   END_IF;
END_REGION

REGION Network 4: CLOSED LOOP FOR THE FLOW EXERCISE 3
   IF "P_Flow3" THEN
       "PID_Compact_5"(Setpoint := "PID_in_SP",   // PID_Compact
                       Input_PER := "VP_Flow",
                       Reset := "start_scada" OR ("PID_in_SP" = 0),
                       Output_PER => "AnOut2_PV");
   END_IF;
END_REGION

REGION Network 5: CLOSED LOOP FOR THE LEVEL EXERCISE 1
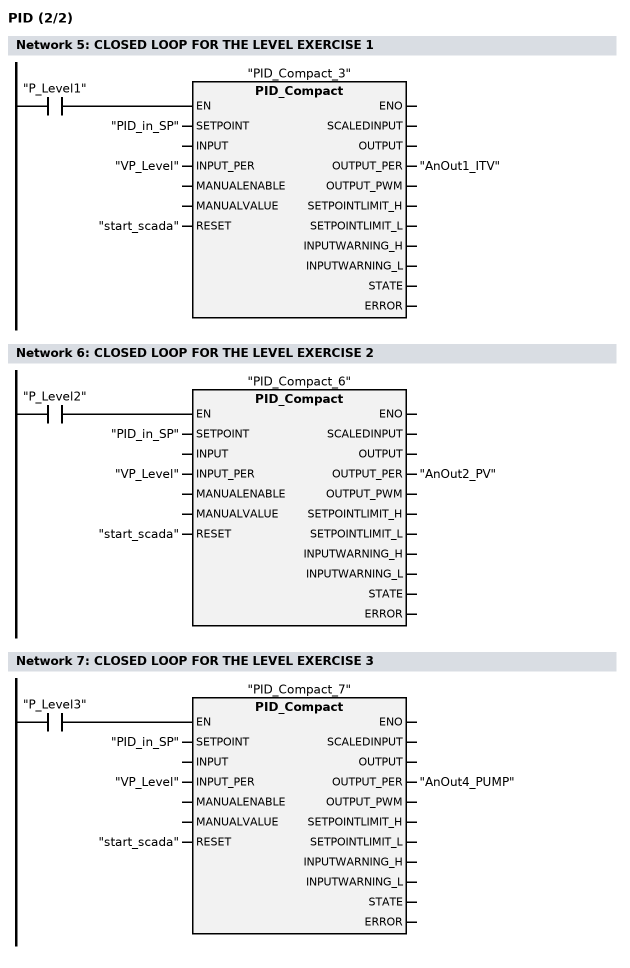
   IF "P_Level1" THEN
       "PID_Compact_3"(Setpoint := "PID_in_SP",   // PID_Compact
                       Input_PER := "VP_Level",
                       Reset := "start_scada",
                       Output_PER => "AnOut1_ITV");
   END_IF;
END_REGION

REGION Network 6: CLOSED LOOP FOR THE LEVEL EXERCISE 2
   IF "P_Level2" THEN
       "PID_Compact_6"(Setpoint := "PID_in_SP",   // PID_Compact
                       Input_PER := "VP_Level",
                       Reset := "start_scada",
                       Output_PER => "AnOut2_PV");
   END_IF;
END_REGION

REGION Network 7: CLOSED LOOP FOR THE LEVEL EXERCISE 3
   IF "P_Level3" THEN
       "PID_Compact_7"(Setpoint := "PID_in_SP",   // PID_Compact
                       Input_PER := "VP_Level",
                       Reset := "start_scada",
                       Output_PER => "AnOut4_PUMP");
   END_IF;
END_REGION
END_ORGANIZATION_BLOCK

// ===== PLC "IPC202B"  CPU 1214C DC/DC/DC =====

VAR_GLOBAL   // PLC tag table "Tabla de variables estándar"
   "start" AT %I0.0 : Bool;   // Start pushbutton
   "stop" AT %I0.1 : Bool;   // Stop pushbutton
   "automan" AT %I0.2 : Bool;   // Automatic/Manual selector
   "reset" AT %I0.3 : Bool;   // Reset pushbutton
   "a0" AT %I0.4 : Bool;   // Plate pusher cylinder backward
   "c0" AT %I0.5 : Bool;   // Unloading manipulator upward
   "c1" AT %I0.6 : Bool;   // Unloading manipulator downward
   "d0" AT %I0.7 : Bool;   // Unloading manipulator backward
   "d1" AT %I1.0 : Bool;   // Unloading manipulator forward
   "e1" AT %I1.1 : Bool;   // Unloading gripper closed
   "f0" AT %I1.2 : Bool;   // Cover feeder cylinders backward
   "f1" AT %I1.3 : Bool;   // Cover feeder cylinders forward
   "g0" AT %I1.4 : Bool;   // Cover pressing cylinder upward
   "g1" AT %I1.5 : Bool;   // Cover pressing cylinder downward
   "h0" AT %I2.0 : Bool;   // Load manipulator downward
   "h1" AT %I2.1 : Bool;   // Load manipulator upward
   "i0" AT %I2.2 : Bool;   // Load manipulator backward
   "i1" AT %I2.3 : Bool;   // Load manipulator forward
   "l1" AT %I2.4 : Bool;   // Can position checker cylinder forward
   "m0" AT %I2.5 : Bool;   // Can pusher cylinder backward
   "m1" AT %I2.6 : Bool;   // Can pusher cylinder forward
   "n0" AT %I2.7 : Bool;   // Can rotary actuator backward
   "n1" AT %I3.0 : Bool;   // Can rotary actuator forward
   "dp1" AT %I3.1 : Bool;   // Can presence at filling position
   "BR" AT %Q0.0 : Bool;   // Red light
   "A+" AT %Q0.1 : Bool;   // Plate pusher cylinder forwards
   "B+" AT %Q0.2 : Bool;   // Lock cylinders of the plate forwards
   "C+" AT %Q0.3 : Bool;   // Unloading manipulator downwards
   "D+" AT %Q0.4 : Bool;   // Unloading manipulator turns
   "E+" AT %Q0.5 : Bool;   // Unloading gripper closure
   "F+" AT %Q0.6 : Bool;   // Lower gripper closure of the covers feeder
   "G+" AT %Q0.7 : Bool;   // Cover pressing cylinder downwards
   "H+" AT %Q1.0 : Bool;   // Load manipulator upwards
   "I+" AT %Q1.1 : Bool;   // Load manipulator forwards
   "J+" AT %Q4.0 : Bool;   // Load gripper closure
   "K+" AT %Q4.1 : Bool;   // Can feeder cylinders forwards
   "L+" AT %Q4.2 : Bool;   // Can position checker cylinder forwards
   "M+" AT %Q4.3 : Bool;   // Can pusher cylinder forwards
   "N+" AT %Q4.4 : Bool;   // Can rotary actuator forwards
   "A4+" AT %Q4.5 : Bool;   // Filling valve opening
   "O+" AT %Q4.6 : Bool;   // Upper gripper closure of the covers feeder
   "step_0" AT %M0.0 : Bool;   // Grafcet first step
   "step_10" AT %M0.1 : Bool;   // Can feeder cylinder forwards
   "step_11" AT %M0.2 : Bool;   // Can position checker cylinder forwards
   "step_12" AT %M0.3 : Bool;   // Can position checker cylinder backwards
   "step_13" AT %M0.4 : Bool;   // Can feeder cylinders backwards
   "step_14" AT %M0.5 : Bool;   // Can pusher cylinder forwards
   "step_15" AT %M0.6 : Bool;   // Can pusher cylinder backwards
   "step_16" AT %M0.7 : Bool;   // Can rotary actuator forwards
   "step_17" AT %M1.0 : Bool;   // Can pusher cylinder forwards
   "step_18" AT %M1.1 : Bool;   // Can pusher cylinder backwards
   "step_19" AT %M1.2 : Bool;   // Can rotary actuator backwards
   "step_20" AT %M1.3 : Bool;   // Loading gripper closure
   "step_21" AT %M1.4 : Bool;   // Loading manipulator upwards
   "step_22" AT %M1.5 : Bool;   // Loading manipulator forwards
   "step_23" AT %M1.6 : Bool;   // Loading manipulator downwards
   "step_24" AT %M1.7 : Bool;   // Loading gripper opening
   "step_25" AT %M2.0 : Bool;   // Loading manipualtor upwards
   "step_26" AT %M2.1 : Bool;   // Loading manipulator backwards
   "step_27" AT %M2.2 : Bool;   // Loading manipualtor downwards
   "step_28" AT %M2.3 : Bool;   // Loading procedure last step
   "step_60" AT %M2.4 : Bool;   // Filling procedure first step
   "step_61" AT %M2.5 : Bool;   // Filling valve opening
   "step_62" AT %M2.6 : Bool;   // Filling valve closure
   "step_63" AT %M2.7 : Bool;   // Filling procedure last step
   "step_40" AT %M3.0 : Bool;   // Pressing procedure first step
   "step_41" AT %M3.1 : Bool;   // Pressing cylinder downwards
   "step_42" AT %M3.2 : Bool;   // Pressing cylinder upwards
   "step_43" AT %M3.3 : Bool;   // Pressing procedure last step
   "step_50" AT %M3.4 : Bool;   // Unloading procedure first step
   "step_51" AT %M3.5 : Bool;   // Unloading manipulator downwards
   "step_52" AT %M3.6 : Bool;   // Unloading gripper closure
   "step_53" AT %M3.7 : Bool;   // Unloading manipualtor upwards
   "step_54" AT %M4.0 : Bool;   // Unloading manipulator forwards
   "step_55" AT %M4.1 : Bool;   // Unloading manipualtor downwards
   "step_56" AT %M4.2 : Bool;   // Unloading gripper opening
   "step_57" AT %M4.3 : Bool;   // Unloading manipualtor upwards
   "step_58" AT %M4.4 : Bool;   // Unloading manipulator backwards
   "step_59" AT %M4.5 : Bool;   // Unloading procedure last step
   "step_70" AT %M4.6 : Bool;   // Red light blinking
   "step_71" AT %M4.7 : Bool;   // Red light off
   "step_1" AT %M5.0 : Bool;   // Plate pusher cylinder forwards
   "step_2" AT %M5.1 : Bool;   // Lock cylinders of the plate forwards
   "step_3" AT %M5.2 : Bool;   // Plate pusher cylinder backwards
   "step_4" AT %M5.3 : Bool;   // Lock cylinders of the plate backwards
   "step_30" AT %M5.4 : Bool;   // Cover feeding procedure first step
   "step_31" AT %M5.5 : Bool;   // Cover feeder cylinders forwards
   "step_32" AT %M5.6 : Bool;   // Cover feeder cylinders backwards
   "step_33" AT %M5.7 : Bool;   // Cover feeding procedure last step
   "positions_can" AT %MW6 : Word;   // Register of the full positions of the plate
   "fill_can" AT %M6.0 : Bool;   // Can at filling position
   "feed_cover_can" AT %M6.1 : Bool;   // Can at cover feeding position
   "press_can" AT %M6.2 : Bool;   // Can at cover pressing position
   "unload_can" AT %M6.3 : Bool;   // Can at unloading position
   "reserved_shl_w_4" AT %M6.4 : Bool;   // Bit 4 of positions register (reserved)
   "reserved_shl_w_5" AT %M6.5 : Bool;   // Bit 5 of positions register (reserved)
   "reserved_shl_w_6" AT %M6.6 : Bool;   // Bit 6 of positions register (reserved)
   "reserved_shl_w_7" AT %M6.7 : Bool;   // Bit 7 of positions register (reserved)
   "reserved_shl_w_8" AT %M7.0 : Bool;   // Bit 8 of positions register (reserved)
   "reserved_shl_w_9" AT %M7.1 : Bool;   // Bit 9 of positions register (reserved)
   "reserved_shl_w_10" AT %M7.2 : Bool;   // Bit 10 of positions register (reserved)
   "reserved_shl_w_11" AT %M7.3 : Bool;   // Bit 11 of positions register (reserved)
   "reserved_shl_w_12" AT %M7.4 : Bool;   // Bit 12 of positions register (reserved)
   "reserved_shl_w_13" AT %M7.5 : Bool;   // Bit 13 of positions register (reserved)
   "reserved_shl_w_14" AT %M7.6 : Bool;   // Bit 14 of positions register (reserved)
   "reserved_shl_w_15" AT %M7.7 : Bool;   // Bit 15 of positions register (reserved)
   "rotate_can_positions" AT %MB8 : Byte;   // Number of positions to rotate
   "reserved_clock_mem_0" AT %M100.0 : Bool;   // Bit 0 of clock
   "reserved_clock_mem_1" AT %M100.1 : Bool;   // Bit 1 of clock
   "reserved_clock_mem_2" AT %M100.2 : Bool;   // Bit 2 of clock
   "reserved_clock_mem_3" AT %M100.3 : Bool;   // Bit 3 of clock
   "reserved_clock_mem_4" AT %M100.4 : Bool;   // Bit 4 of clock
   "clock_1_second" AT %M100.5 : Bool;   // 1 second period clock
   "reserved_clock_mem_6" AT %M100.6 : Bool;   // Bit 6 of clock
   "reserved_clock_mem_7" AT %M100.7 : Bool;   // Bit 7 of clock
   "continue" AT %M9.0 : Bool;   // Continue program sequence
   "auto" AT %M9.1 : Bool;   // Automatic mode of the station
   "initial_conditions" AT %M9.2 : Bool;   // Initial conditions of the station
   "check_ok" AT %M9.3 : Bool;   // Properly positioned can verification
   "unloading_cycle" AT %M9.4 : Bool;   // Unloading cycle done indication
   "memory_bit_step_2" AT %M9.5 : Bool;   // Bit memory of step 2
   "Clock_Byte" AT %MB100 : Byte;
   "IPC1_on" AT %I10.0 : Bool;   // IPC201C active
   "IPC1_end" AT %I10.1 : Bool;   // End cycle of IPC201C
   "IPC1_full" AT %I10.2 : Bool;   // Central tank full in IPC201C
   "start_scada" AT %M10.0 : Bool;   // Start from the SCADA // PC --> PLC
   "stop_scada" AT %M10.1 : Bool;   // Stop from the SCADA // PC --> PLC
   "reset_scada" AT %M10.3 : Bool;   // Reset from the SCADA // PC --> PLC
   "automan_scada" AT %M10.2 : Bool;   // Auto/Man from the SCADA // PC --> PLC
   "IPC2_on" AT %Q10.0 : Bool;   // IPC202 active
   "IPC3_start_cycle" AT %Q10.2 : Bool;   // Start cycle to IPC203
   "Output_channel_0" AT %MB20 : Byte;   // Output channel 0 to SCADA // PLC --> PC
   "Output_channel_1" AT %MB21 : Byte;   // Output channel 1 to SCADA // PLC --> PC
   "Output_channel_2" AT %MB22 : Byte;   // Output channel 2 to SCADA // PLC --> PC
   "Output_channel_3" AT %MB23 : Byte;   // Output channel 3 to SCADA // PLC --> PC
   "Output_channel_4" AT %MB24 : Byte;   // Output channel 4 to SCADA // PLC --> PC
   "Output_channel_5" AT %MB25 : Byte;   // Output channel 5 to SCADA // PLC --> PC
   "Output_channel_6" AT %MB26 : Byte;   // Output channel 6 to SCADA // PLC --> PC
   "Input_0" AT %IB0 : Byte;   // Physical inputs channel 0
   "Input_1" AT %IB1 : Byte;   // Physical inputs channel 1
   "Input_2" AT %IB2 : Byte;   // Physical inputs channel 2
   "Input_3" AT %IB3 : Byte;   // Physical inputs channel 3
   "Output_0" AT %QB0 : Byte;   // Physical outputs channel 0
   "Output_1" AT %QB1 : Byte;   // Physical outputs channel 1
   "Output_2" AT %QB4 : Byte;   // Physical outputs channel 2
   "Output_channel_7" AT %MW27 : Word;   // Output channel 7 to SCADA // PLC --> PC
   "IPC3_on" AT %I20.0 : Bool;   // IPC3 active
   "IPC3_end" AT %I20.1 : Bool;   // End cycle of IPC3
   "IPC3_dp1" AT %I20.2 : Bool;   // Can presence in IPC203
   "IPC1_start_cycle" AT %Q10.1 : Bool;   // Start cycle to IPC201
   "Tag_2" AT %QB10 : Byte;
   "Tag_3" AT %M105.3 : Bool;
END_VAR

// folder: System blocks/Program resources

DATA_BLOCK "Timer_0"   // DB1
{ S7_Optimized_Access := 'TRUE' }
AUTHOR : Simatic
FAMILY : IEC
NAME : IEC_TMR
VERSION : 1.0
// stored: InstanceOfName IEC_TIMER
"IEC_TIMER"
BEGIN
END_DATA_BLOCK

DATA_BLOCK "Timer_1"   // DB2
{ S7_Optimized_Access := 'TRUE' }
AUTHOR : Simatic
FAMILY : IEC
NAME : IEC_TMR
VERSION : 1.0
// stored: InstanceOfName IEC_TIMER
"IEC_TIMER"
BEGIN
END_DATA_BLOCK

DATA_BLOCK "Timer_2"   // DB3
{ S7_Optimized_Access := 'TRUE' }
AUTHOR : Simatic
FAMILY : IEC
NAME : IEC_TMR
VERSION : 1.0
// stored: InstanceOfName IEC_TIMER
"IEC_TIMER"
BEGIN
END_DATA_BLOCK

DATA_BLOCK "Timer_3"   // DB4
{ S7_Optimized_Access := 'TRUE' }
AUTHOR : Simatic
FAMILY : IEC
NAME : IEC_TMR
VERSION : 1.0
// stored: InstanceOfName IEC_TIMER
"IEC_TIMER"
BEGIN
END_DATA_BLOCK

DATA_BLOCK "Timer_4"   // DB5
{ S7_Optimized_Access := 'TRUE' }
AUTHOR : Simatic
FAMILY : IEC
NAME : IEC_TMR
VERSION : 1.0
// stored: InstanceOfName IEC_TIMER
"IEC_TIMER"
BEGIN
END_DATA_BLOCK

DATA_BLOCK "Timer_5"   // DB6
{ S7_Optimized_Access := 'TRUE' }
AUTHOR : Simatic
FAMILY : IEC
NAME : IEC_TMR
VERSION : 1.0
// stored: InstanceOfName IEC_TIMER
"IEC_TIMER"
BEGIN
END_DATA_BLOCK

DATA_BLOCK "Timer_6"   // DB7
{ S7_Optimized_Access := 'TRUE' }
AUTHOR : Simatic
FAMILY : IEC
NAME : IEC_TMR
VERSION : 1.0
// stored: InstanceOfName IEC_TIMER
"IEC_TIMER"
BEGIN
END_DATA_BLOCK

DATA_BLOCK "Timer_7"   // DB8
{ S7_Optimized_Access := 'TRUE' }
AUTHOR : Simatic
FAMILY : IEC
NAME : IEC_TMR
VERSION : 1.0
// stored: InstanceOfName IEC_TIMER
"IEC_TIMER"
BEGIN
END_DATA_BLOCK

DATA_BLOCK "Timer_8"   // DB9
{ S7_Optimized_Access := 'TRUE' }
AUTHOR : Simatic
FAMILY : IEC
NAME : IEC_TMR
VERSION : 1.0
// stored: InstanceOfName IEC_TIMER
"IEC_TIMER"
BEGIN
END_DATA_BLOCK

DATA_BLOCK "Timer_9"   // DB10
{ S7_Optimized_Access := 'TRUE' }
AUTHOR : Simatic
FAMILY : IEC
NAME : IEC_TMR
VERSION : 1.0
// stored: InstanceOfName IEC_TIMER
"IEC_TIMER"
BEGIN
END_DATA_BLOCK

DATA_BLOCK "Timer_10"   // DB11
{ S7_Optimized_Access := 'TRUE' }
AUTHOR : Simatic
FAMILY : IEC
NAME : IEC_TMR
VERSION : 1.0
// stored: InstanceOfName IEC_TIMER
"IEC_TIMER"
BEGIN
END_DATA_BLOCK

DATA_BLOCK "Timer_11"   // DB12
{ S7_Optimized_Access := 'TRUE' }
AUTHOR : Simatic
FAMILY : IEC
NAME : IEC_TMR
VERSION : 1.0
// stored: InstanceOfName IEC_TIMER
"IEC_TIMER"
BEGIN
END_DATA_BLOCK

DATA_BLOCK "Timer_12"   // DB13
{ S7_Optimized_Access := 'TRUE' }
AUTHOR : Simatic
FAMILY : IEC
NAME : IEC_TMR
VERSION : 1.0
// stored: InstanceOfName IEC_TIMER
"IEC_TIMER"
BEGIN
END_DATA_BLOCK

DATA_BLOCK "Timer_13"   // DB14
{ S7_Optimized_Access := 'TRUE' }
AUTHOR : Simatic
FAMILY : IEC
NAME : IEC_TMR
VERSION : 1.0
// stored: InstanceOfName IEC_TIMER
"IEC_TIMER"
BEGIN
END_DATA_BLOCK

DATA_BLOCK "Timer_14"   // DB15
{ S7_Optimized_Access := 'TRUE' }
AUTHOR : Simatic
FAMILY : IEC
NAME : IEC_TMR
VERSION : 1.0
// stored: InstanceOfName IEC_TIMER
"IEC_TIMER"
BEGIN
END_DATA_BLOCK

DATA_BLOCK "Timer_15"   // DB16
{ S7_Optimized_Access := 'TRUE' }
AUTHOR : Simatic
FAMILY : IEC
NAME : IEC_TMR
VERSION : 1.0
// stored: InstanceOfName IEC_TIMER
"IEC_TIMER"
BEGIN
END_DATA_BLOCK

DATA_BLOCK "Timer_16"   // DB17
{ S7_Optimized_Access := 'TRUE' }
AUTHOR : Simatic
FAMILY : IEC
NAME : IEC_TMR
VERSION : 1.0
// stored: InstanceOfName IEC_TIMER
"IEC_TIMER"
BEGIN
END_DATA_BLOCK

DATA_BLOCK "Timer_17"   // DB18
{ S7_Optimized_Access := 'TRUE' }
AUTHOR : Simatic
FAMILY : IEC
NAME : IEC_TMR
VERSION : 1.0
// stored: InstanceOfName IEC_TIMER
"IEC_TIMER"
BEGIN
END_DATA_BLOCK

DATA_BLOCK "Timer_18"   // DB19
{ S7_Optimized_Access := 'TRUE' }
AUTHOR : Simatic
FAMILY : IEC
NAME : IEC_TMR
VERSION : 1.0
// stored: InstanceOfName IEC_TIMER
"IEC_TIMER"
BEGIN
END_DATA_BLOCK

DATA_BLOCK "Timer_19"   // DB20
{ S7_Optimized_Access := 'TRUE' }
AUTHOR : Simatic
FAMILY : IEC
NAME : IEC_TMR
VERSION : 1.0
// stored: InstanceOfName IEC_TIMER
"IEC_TIMER"
BEGIN
END_DATA_BLOCK

DATA_BLOCK "Timer_20"   // DB21
{ S7_Optimized_Access := 'TRUE' }
AUTHOR : Simatic
FAMILY : IEC
NAME : IEC_TMR
VERSION : 1.0
// stored: InstanceOfName IEC_TIMER
"IEC_TIMER"
BEGIN
END_DATA_BLOCK

DATA_BLOCK "Timer_21"   // DB22
{ S7_Optimized_Access := 'TRUE' }
AUTHOR : Simatic
FAMILY : IEC
NAME : IEC_TMR
VERSION : 1.0
// stored: InstanceOfName IEC_TIMER
"IEC_TIMER"
BEGIN
END_DATA_BLOCK

DATA_BLOCK "Timer_22"   // DB23
{ S7_Optimized_Access := 'TRUE' }
AUTHOR : Simatic
FAMILY : IEC
NAME : IEC_TMR
VERSION : 1.0
// stored: InstanceOfName IEC_TIMER
"IEC_TIMER"
BEGIN
END_DATA_BLOCK

DATA_BLOCK "Timer_23"   // DB24
{ S7_Optimized_Access := 'TRUE' }
AUTHOR : Simatic
FAMILY : IEC
NAME : IEC_TMR
VERSION : 1.0
// stored: InstanceOfName IEC_TIMER
"IEC_TIMER"
BEGIN
END_DATA_BLOCK

DATA_BLOCK "Timer_24"   // DB25
{ S7_Optimized_Access := 'TRUE' }
AUTHOR : Simatic
FAMILY : IEC
NAME : IEC_TMR
VERSION : 1.0
// stored: InstanceOfName IEC_TIMER
"IEC_TIMER"
BEGIN
END_DATA_BLOCK

DATA_BLOCK "Timer_25"   // DB26
{ S7_Optimized_Access := 'TRUE' }
AUTHOR : Simatic
FAMILY : IEC
NAME : IEC_TMR
VERSION : 1.0
// stored: InstanceOfName IEC_TIMER
"IEC_TIMER"
BEGIN
END_DATA_BLOCK

DATA_BLOCK "Timer_26"   // DB27
{ S7_Optimized_Access := 'TRUE' }
AUTHOR : Simatic
FAMILY : IEC
NAME : IEC_TMR
VERSION : 1.0
// stored: InstanceOfName IEC_TIMER
"IEC_TIMER"
BEGIN
END_DATA_BLOCK

DATA_BLOCK "Timer_27"   // DB28
{ S7_Optimized_Access := 'TRUE' }
AUTHOR : Simatic
FAMILY : IEC
NAME : IEC_TMR
VERSION : 1.0
// stored: InstanceOfName IEC_TIMER
"IEC_TIMER"
BEGIN
END_DATA_BLOCK

DATA_BLOCK "Timer_28"   // DB29
{ S7_Optimized_Access := 'TRUE' }
AUTHOR : Simatic
FAMILY : IEC
NAME : IEC_TMR
VERSION : 1.0
// stored: InstanceOfName IEC_TIMER
"IEC_TIMER"
BEGIN
END_DATA_BLOCK

// folder: (top level)

FUNCTION "STEPS" : Void   // FC1, LAD
TITLE = STEPS
{ S7_Optimized_Access := 'TRUE' }
VERSION : 0.1
BEGIN

REGION Network 1: GRAFCET first step
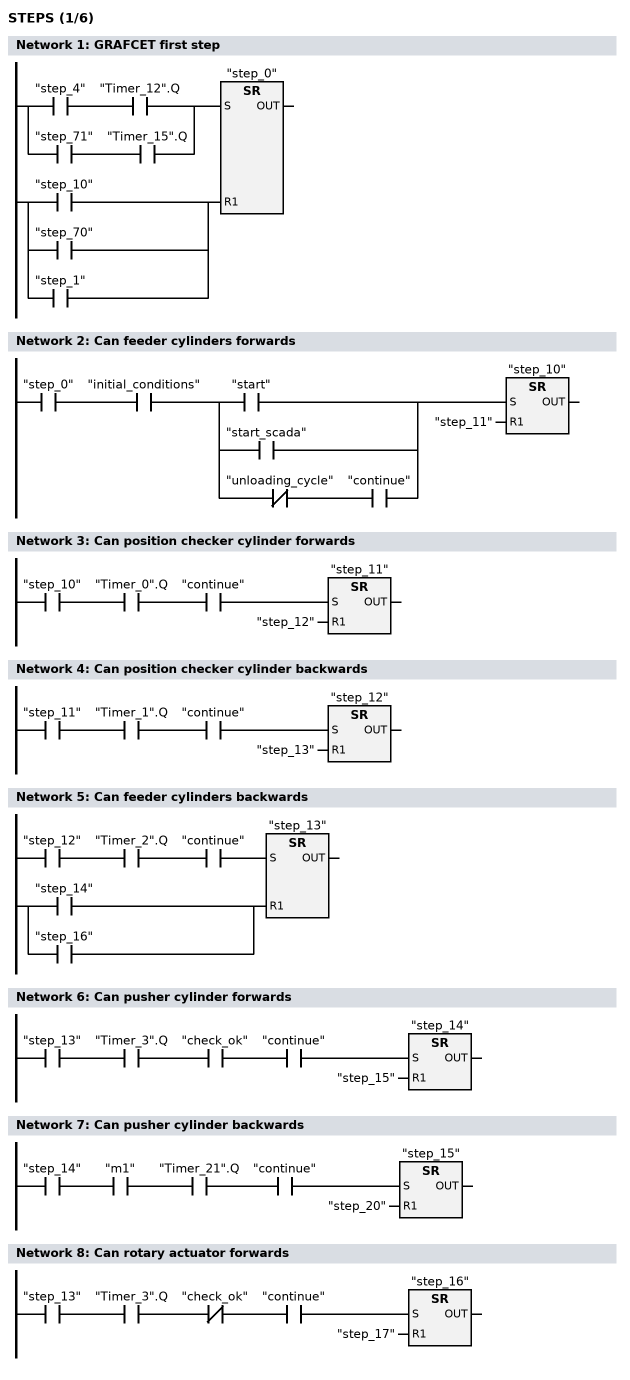
   RUNG wire#powerrail
      Contact( "step_4" )
      Contact( "Timer_12".Q )
      wire#w1
      S_SR(operand := "step_0", r1 := wire#w2)
   END_RUNG
   RUNG wire#powerrail
      Contact( "step_71" )
      Contact( "Timer_15".Q )
   END_RUNG wire#w1
   RUNG wire#powerrail
      Contact( "step_10" )
   END_RUNG wire#w2
   RUNG wire#powerrail
      Contact( "step_70" )
   END_RUNG wire#w2
   RUNG wire#powerrail
      Contact( "step_1" )
   END_RUNG wire#w2
   // the same network as SCL:
   IF ("step_4" AND "Timer_12".Q) OR ("step_71" AND "Timer_15".Q) THEN
       "step_0" := TRUE;   // SR flip-flop
   END_IF;
   IF "step_10" OR "step_70" OR "step_1" THEN "step_0" := FALSE; END_IF;
END_REGION

REGION Network 2: Can feeder cylinders forwards
   RUNG wire#powerrail
      Contact( "step_0" )
      Contact( "initial_conditions" )
      wire#w1
      Contact( "start" )
      wire#w2
      S_SR(operand := "step_10", r1 := "step_11")
   END_RUNG
   RUNG wire#w1
      Contact( "start_scada" )
   END_RUNG wire#w2
   RUNG wire#w1
      I_Contact( "unloading_cycle" )
      Contact( "continue" )
   END_RUNG wire#w2
   // the same network as SCL:
   IF "step_0" AND "initial_conditions" AND ("start" OR "start_scada" OR (NOT "unloading_cycle" AND "continue")) THEN
       "step_10" := TRUE;   // SR flip-flop
   END_IF;
   IF "step_11" THEN "step_10" := FALSE; END_IF;
END_REGION

REGION Network 3: Can position checker cylinder forwards
   RUNG wire#powerrail
      Contact( "step_10" )
      Contact( "Timer_0".Q )
      Contact( "continue" )
      S_SR(operand := "step_11", r1 := "step_12")
   END_RUNG
   // the same network as SCL:
   IF "step_10" AND "Timer_0".Q AND "continue" THEN
       "step_11" := TRUE;   // SR flip-flop
   END_IF;
   IF "step_12" THEN "step_11" := FALSE; END_IF;
END_REGION

REGION Network 4: Can position checker cylinder backwards
   RUNG wire#powerrail
      Contact( "step_11" )
      Contact( "Timer_1".Q )
      Contact( "continue" )
      S_SR(operand := "step_12", r1 := "step_13")
   END_RUNG
   // the same network as SCL:
   IF "step_11" AND "Timer_1".Q AND "continue" THEN
       "step_12" := TRUE;   // SR flip-flop
   END_IF;
   IF "step_13" THEN "step_12" := FALSE; END_IF;
END_REGION

REGION Network 5: Can feeder cylinders backwards
   RUNG wire#powerrail
      Contact( "step_12" )
      Contact( "Timer_2".Q )
      Contact( "continue" )
      S_SR(operand := "step_13", r1 := wire#w1)
   END_RUNG
   RUNG wire#powerrail
      Contact( "step_14" )
   END_RUNG wire#w1
   RUNG wire#powerrail
      Contact( "step_16" )
   END_RUNG wire#w1
   // the same network as SCL:
   IF "step_12" AND "Timer_2".Q AND "continue" THEN
       "step_13" := TRUE;   // SR flip-flop
   END_IF;
   IF "step_14" OR "step_16" THEN "step_13" := FALSE; END_IF;
END_REGION

REGION Network 6: Can pusher cylinder forwards
   RUNG wire#powerrail
      Contact( "step_13" )
      Contact( "Timer_3".Q )
      Contact( "check_ok" )
      Contact( "continue" )
      S_SR(operand := "step_14", r1 := "step_15")
   END_RUNG
   // the same network as SCL:
   IF "step_13" AND "Timer_3".Q AND "check_ok" AND "continue" THEN
       "step_14" := TRUE;   // SR flip-flop
   END_IF;
   IF "step_15" THEN "step_14" := FALSE; END_IF;
END_REGION

REGION Network 7: Can pusher cylinder backwards
   RUNG wire#powerrail
      Contact( "step_14" )
      Contact( "m1" )
      Contact( "Timer_21".Q )
      Contact( "continue" )
      S_SR(operand := "step_15", r1 := "step_20")
   END_RUNG
   // the same network as SCL:
   IF "step_14" AND "m1" AND "Timer_21".Q AND "continue" THEN
       "step_15" := TRUE;   // SR flip-flop
   END_IF;
   IF "step_20" THEN "step_15" := FALSE; END_IF;
END_REGION

REGION Network 8: Can rotary actuator forwards
   RUNG wire#powerrail
      Contact( "step_13" )
      Contact( "Timer_3".Q )
      I_Contact( "check_ok" )
      Contact( "continue" )
      S_SR(operand := "step_16", r1 := "step_17")
   END_RUNG
   // the same network as SCL:
   IF "step_13" AND "Timer_3".Q AND NOT "check_ok" AND "continue" THEN
       "step_16" := TRUE;   // SR flip-flop
   END_IF;
   IF "step_17" THEN "step_16" := FALSE; END_IF;
END_REGION

REGION Network 9: Can pusher cylinder forwards
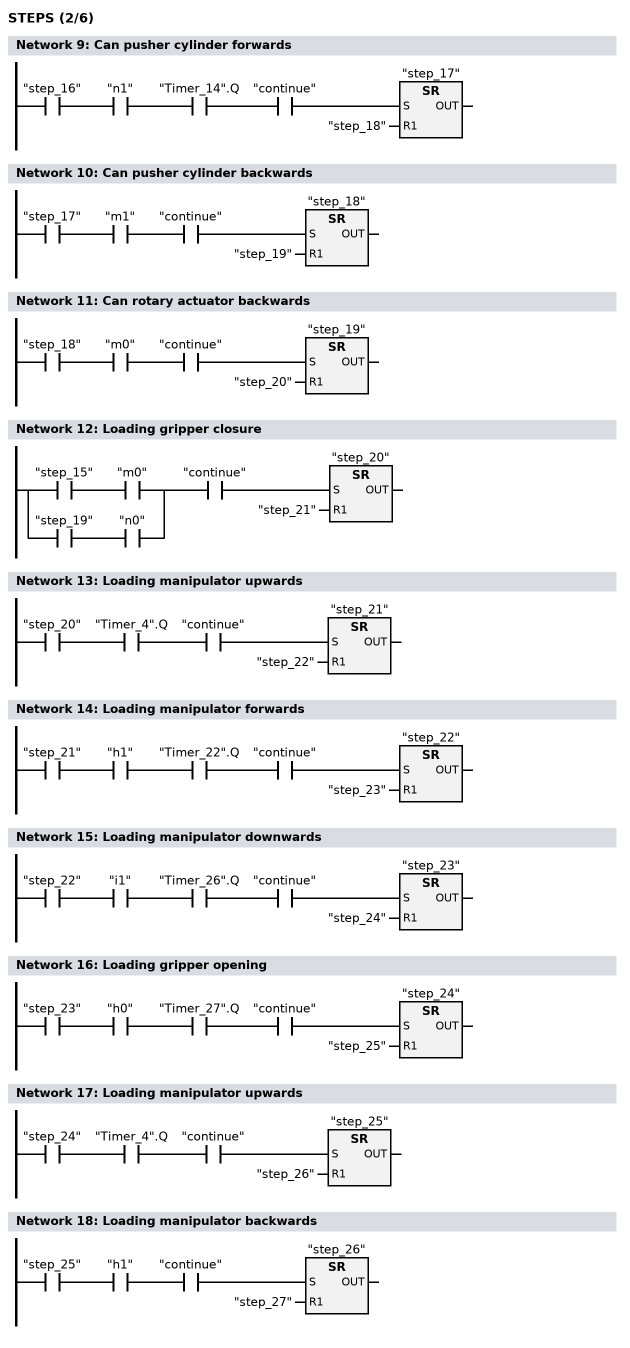
   RUNG wire#powerrail
      Contact( "step_16" )
      Contact( "n1" )
      Contact( "Timer_14".Q )
      Contact( "continue" )
      S_SR(operand := "step_17", r1 := "step_18")
   END_RUNG
   // the same network as SCL:
   IF "step_16" AND "n1" AND "Timer_14".Q AND "continue" THEN
       "step_17" := TRUE;   // SR flip-flop
   END_IF;
   IF "step_18" THEN "step_17" := FALSE; END_IF;
END_REGION

REGION Network 10: Can pusher cylinder backwards
   RUNG wire#powerrail
      Contact( "step_17" )
      Contact( "m1" )
      Contact( "continue" )
      S_SR(operand := "step_18", r1 := "step_19")
   END_RUNG
   // the same network as SCL:
   IF "step_17" AND "m1" AND "continue" THEN
       "step_18" := TRUE;   // SR flip-flop
   END_IF;
   IF "step_19" THEN "step_18" := FALSE; END_IF;
END_REGION

REGION Network 11: Can rotary actuator backwards
   RUNG wire#powerrail
      Contact( "step_18" )
      Contact( "m0" )
      Contact( "continue" )
      S_SR(operand := "step_19", r1 := "step_20")
   END_RUNG
   // the same network as SCL:
   IF "step_18" AND "m0" AND "continue" THEN
       "step_19" := TRUE;   // SR flip-flop
   END_IF;
   IF "step_20" THEN "step_19" := FALSE; END_IF;
END_REGION

REGION Network 12: Loading gripper closure
   RUNG wire#powerrail
      Contact( "step_15" )
      Contact( "m0" )
      wire#w1
      Contact( "continue" )
      S_SR(operand := "step_20", r1 := "step_21")
   END_RUNG
   RUNG wire#powerrail
      Contact( "step_19" )
      Contact( "n0" )
   END_RUNG wire#w1
   // the same network as SCL:
   IF (("step_15" AND "m0") OR ("step_19" AND "n0")) AND "continue" THEN
       "step_20" := TRUE;   // SR flip-flop
   END_IF;
   IF "step_21" THEN "step_20" := FALSE; END_IF;
END_REGION

REGION Network 13: Loading manipulator upwards
   RUNG wire#powerrail
      Contact( "step_20" )
      Contact( "Timer_4".Q )
      Contact( "continue" )
      S_SR(operand := "step_21", r1 := "step_22")
   END_RUNG
   // the same network as SCL:
   IF "step_20" AND "Timer_4".Q AND "continue" THEN
       "step_21" := TRUE;   // SR flip-flop
   END_IF;
   IF "step_22" THEN "step_21" := FALSE; END_IF;
END_REGION

REGION Network 14: Loading manipulator forwards
   RUNG wire#powerrail
      Contact( "step_21" )
      Contact( "h1" )
      Contact( "Timer_22".Q )
      Contact( "continue" )
      S_SR(operand := "step_22", r1 := "step_23")
   END_RUNG
   // the same network as SCL:
   IF "step_21" AND "h1" AND "Timer_22".Q AND "continue" THEN
       "step_22" := TRUE;   // SR flip-flop
   END_IF;
   IF "step_23" THEN "step_22" := FALSE; END_IF;
END_REGION

REGION Network 15: Loading manipulator downwards
   RUNG wire#powerrail
      Contact( "step_22" )
      Contact( "i1" )
      Contact( "Timer_26".Q )
      Contact( "continue" )
      S_SR(operand := "step_23", r1 := "step_24")
   END_RUNG
   // the same network as SCL:
   IF "step_22" AND "i1" AND "Timer_26".Q AND "continue" THEN
       "step_23" := TRUE;   // SR flip-flop
   END_IF;
   IF "step_24" THEN "step_23" := FALSE; END_IF;
END_REGION

REGION Network 16: Loading gripper opening
   RUNG wire#powerrail
      Contact( "step_23" )
      Contact( "h0" )
      Contact( "Timer_27".Q )
      Contact( "continue" )
      S_SR(operand := "step_24", r1 := "step_25")
   END_RUNG
   // the same network as SCL:
   IF "step_23" AND "h0" AND "Timer_27".Q AND "continue" THEN
       "step_24" := TRUE;   // SR flip-flop
   END_IF;
   IF "step_25" THEN "step_24" := FALSE; END_IF;
END_REGION

REGION Network 17: Loading manipulator upwards
   RUNG wire#powerrail
      Contact( "step_24" )
      Contact( "Timer_4".Q )
      Contact( "continue" )
      S_SR(operand := "step_25", r1 := "step_26")
   END_RUNG
   // the same network as SCL:
   IF "step_24" AND "Timer_4".Q AND "continue" THEN
       "step_25" := TRUE;   // SR flip-flop
   END_IF;
   IF "step_26" THEN "step_25" := FALSE; END_IF;
END_REGION

REGION Network 18: Loading manipulator backwards
   RUNG wire#powerrail
      Contact( "step_25" )
      Contact( "h1" )
      Contact( "continue" )
      S_SR(operand := "step_26", r1 := "step_27")
   END_RUNG
   // the same network as SCL:
   IF "step_25" AND "h1" AND "continue" THEN
       "step_26" := TRUE;   // SR flip-flop
   END_IF;
   IF "step_27" THEN "step_26" := FALSE; END_IF;
END_REGION

REGION Network 19: Loading manipulator downwards
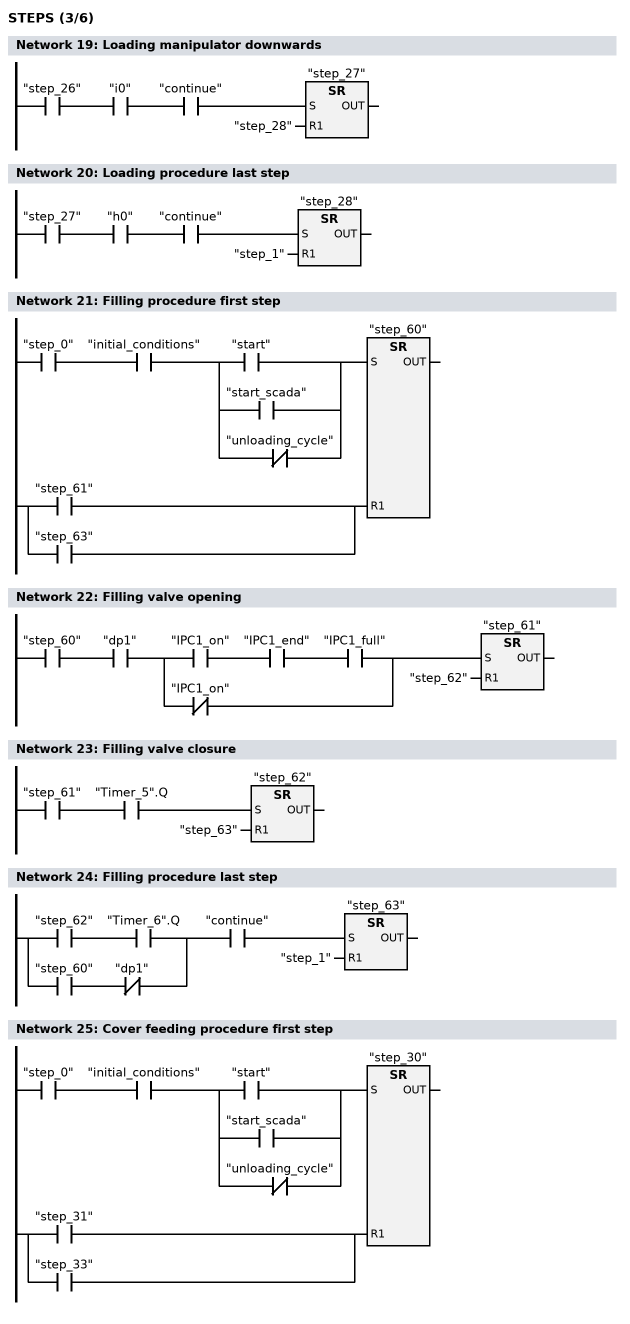
   RUNG wire#powerrail
      Contact( "step_26" )
      Contact( "i0" )
      Contact( "continue" )
      S_SR(operand := "step_27", r1 := "step_28")
   END_RUNG
   // the same network as SCL:
   IF "step_26" AND "i0" AND "continue" THEN
       "step_27" := TRUE;   // SR flip-flop
   END_IF;
   IF "step_28" THEN "step_27" := FALSE; END_IF;
END_REGION

REGION Network 20: Loading procedure last step
   RUNG wire#powerrail
      Contact( "step_27" )
      Contact( "h0" )
      Contact( "continue" )
      S_SR(operand := "step_28", r1 := "step_1")
   END_RUNG
   // the same network as SCL:
   IF "step_27" AND "h0" AND "continue" THEN
       "step_28" := TRUE;   // SR flip-flop
   END_IF;
   IF "step_1" THEN "step_28" := FALSE; END_IF;
END_REGION

REGION Network 21: Filling procedure first step
   RUNG wire#powerrail
      Contact( "step_0" )
      Contact( "initial_conditions" )
      wire#w1
      Contact( "start" )
      wire#w2
      S_SR(operand := "step_60", r1 := wire#w3)
   END_RUNG
   RUNG wire#w1
      Contact( "start_scada" )
   END_RUNG wire#w2
   RUNG wire#w1
      I_Contact( "unloading_cycle" )
   END_RUNG wire#w2
   RUNG wire#powerrail
      Contact( "step_61" )
   END_RUNG wire#w3
   RUNG wire#powerrail
      Contact( "step_63" )
   END_RUNG wire#w3
   // the same network as SCL:
   IF "step_0" AND "initial_conditions" AND ("start" OR "start_scada" OR NOT "unloading_cycle") THEN
       "step_60" := TRUE;   // SR flip-flop
   END_IF;
   IF "step_61" OR "step_63" THEN "step_60" := FALSE; END_IF;
END_REGION

REGION Network 22: Filling valve opening
   RUNG wire#powerrail
      Contact( "step_60" )
      Contact( "dp1" )
      wire#w1
      Contact( "IPC1_on" )
      Contact( "IPC1_end" )
      Contact( "IPC1_full" )
      wire#w2
      S_SR(operand := "step_61", r1 := "step_62")
   END_RUNG
   RUNG wire#w1
      I_Contact( "IPC1_on" )
   END_RUNG wire#w2
   // the same network as SCL:
   IF "step_60" AND "dp1" AND (("IPC1_on" AND "IPC1_end" AND "IPC1_full") OR NOT "IPC1_on") THEN
       "step_61" := TRUE;   // SR flip-flop
   END_IF;
   IF "step_62" THEN "step_61" := FALSE; END_IF;
END_REGION

REGION Network 23: Filling valve closure
   RUNG wire#powerrail
      Contact( "step_61" )
      Contact( "Timer_5".Q )
      S_SR(operand := "step_62", r1 := "step_63")
   END_RUNG
   // the same network as SCL:
   IF "step_61" AND "Timer_5".Q THEN
       "step_62" := TRUE;   // SR flip-flop
   END_IF;
   IF "step_63" THEN "step_62" := FALSE; END_IF;
END_REGION

REGION Network 24: Filling procedure last step
   RUNG wire#powerrail
      Contact( "step_62" )
      Contact( "Timer_6".Q )
      wire#w1
      Contact( "continue" )
      S_SR(operand := "step_63", r1 := "step_1")
   END_RUNG
   RUNG wire#powerrail
      Contact( "step_60" )
      I_Contact( "dp1" )
   END_RUNG wire#w1
   // the same network as SCL:
   IF (("step_62" AND "Timer_6".Q) OR ("step_60" AND NOT "dp1")) AND "continue" THEN
       "step_63" := TRUE;   // SR flip-flop
   END_IF;
   IF "step_1" THEN "step_63" := FALSE; END_IF;
END_REGION

REGION Network 25: Cover feeding procedure first step
   RUNG wire#powerrail
      Contact( "step_0" )
      Contact( "initial_conditions" )
      wire#w1
      Contact( "start" )
      wire#w2
      S_SR(operand := "step_30", r1 := wire#w3)
   END_RUNG
   RUNG wire#w1
      Contact( "start_scada" )
   END_RUNG wire#w2
   RUNG wire#w1
      I_Contact( "unloading_cycle" )
   END_RUNG wire#w2
   RUNG wire#powerrail
      Contact( "step_31" )
   END_RUNG wire#w3
   RUNG wire#powerrail
      Contact( "step_33" )
   END_RUNG wire#w3
   // the same network as SCL:
   IF "step_0" AND "initial_conditions" AND ("start" OR "start_scada" OR NOT "unloading_cycle") THEN
       "step_30" := TRUE;   // SR flip-flop
   END_IF;
   IF "step_31" OR "step_33" THEN "step_30" := FALSE; END_IF;
END_REGION

REGION Network 26: Cover feeder cylinders forwards
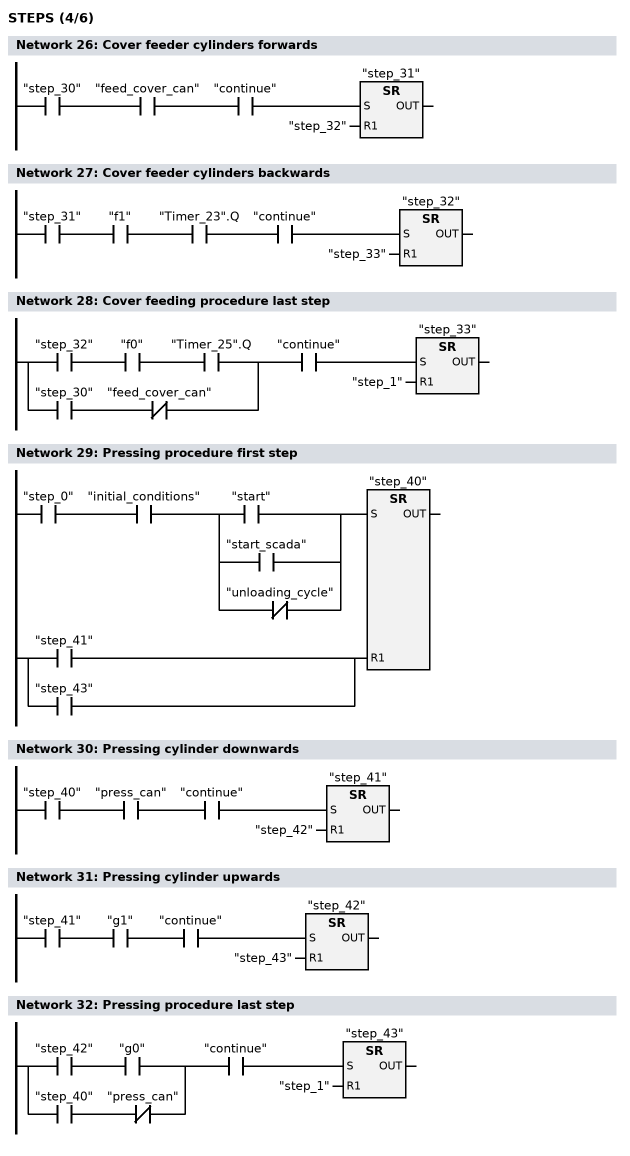
   RUNG wire#powerrail
      Contact( "step_30" )
      Contact( "feed_cover_can" )
      Contact( "continue" )
      S_SR(operand := "step_31", r1 := "step_32")
   END_RUNG
   // the same network as SCL:
   IF "step_30" AND "feed_cover_can" AND "continue" THEN
       "step_31" := TRUE;   // SR flip-flop
   END_IF;
   IF "step_32" THEN "step_31" := FALSE; END_IF;
END_REGION

REGION Network 27: Cover feeder cylinders backwards
   RUNG wire#powerrail
      Contact( "step_31" )
      Contact( "f1" )
      Contact( "Timer_23".Q )
      Contact( "continue" )
      S_SR(operand := "step_32", r1 := "step_33")
   END_RUNG
   // the same network as SCL:
   IF "step_31" AND "f1" AND "Timer_23".Q AND "continue" THEN
       "step_32" := TRUE;   // SR flip-flop
   END_IF;
   IF "step_33" THEN "step_32" := FALSE; END_IF;
END_REGION

REGION Network 28: Cover feeding procedure last step
   RUNG wire#powerrail
      Contact( "step_32" )
      Contact( "f0" )
      Contact( "Timer_25".Q )
      wire#w1
      Contact( "continue" )
      S_SR(operand := "step_33", r1 := "step_1")
   END_RUNG
   RUNG wire#powerrail
      Contact( "step_30" )
      I_Contact( "feed_cover_can" )
   END_RUNG wire#w1
   // the same network as SCL:
   IF (("step_32" AND "f0" AND "Timer_25".Q) OR ("step_30" AND NOT "feed_cover_can")) AND "continue" THEN
       "step_33" := TRUE;   // SR flip-flop
   END_IF;
   IF "step_1" THEN "step_33" := FALSE; END_IF;
END_REGION

REGION Network 29: Pressing procedure first step
   RUNG wire#powerrail
      Contact( "step_0" )
      Contact( "initial_conditions" )
      wire#w1
      Contact( "start" )
      wire#w2
      S_SR(operand := "step_40", r1 := wire#w3)
   END_RUNG
   RUNG wire#w1
      Contact( "start_scada" )
   END_RUNG wire#w2
   RUNG wire#w1
      I_Contact( "unloading_cycle" )
   END_RUNG wire#w2
   RUNG wire#powerrail
      Contact( "step_41" )
   END_RUNG wire#w3
   RUNG wire#powerrail
      Contact( "step_43" )
   END_RUNG wire#w3
   // the same network as SCL:
   IF "step_0" AND "initial_conditions" AND ("start" OR "start_scada" OR NOT "unloading_cycle") THEN
       "step_40" := TRUE;   // SR flip-flop
   END_IF;
   IF "step_41" OR "step_43" THEN "step_40" := FALSE; END_IF;
END_REGION

REGION Network 30: Pressing cylinder downwards
   RUNG wire#powerrail
      Contact( "step_40" )
      Contact( "press_can" )
      Contact( "continue" )
      S_SR(operand := "step_41", r1 := "step_42")
   END_RUNG
   // the same network as SCL:
   IF "step_40" AND "press_can" AND "continue" THEN
       "step_41" := TRUE;   // SR flip-flop
   END_IF;
   IF "step_42" THEN "step_41" := FALSE; END_IF;
END_REGION

REGION Network 31: Pressing cylinder upwards
   RUNG wire#powerrail
      Contact( "step_41" )
      Contact( "g1" )
      Contact( "continue" )
      S_SR(operand := "step_42", r1 := "step_43")
   END_RUNG
   // the same network as SCL:
   IF "step_41" AND "g1" AND "continue" THEN
       "step_42" := TRUE;   // SR flip-flop
   END_IF;
   IF "step_43" THEN "step_42" := FALSE; END_IF;
END_REGION

REGION Network 32: Pressing procedure last step
   RUNG wire#powerrail
      Contact( "step_42" )
      Contact( "g0" )
      wire#w1
      Contact( "continue" )
      S_SR(operand := "step_43", r1 := "step_1")
   END_RUNG
   RUNG wire#powerrail
      Contact( "step_40" )
      I_Contact( "press_can" )
   END_RUNG wire#w1
   // the same network as SCL:
   IF (("step_42" AND "g0") OR ("step_40" AND NOT "press_can")) AND "continue" THEN
       "step_43" := TRUE;   // SR flip-flop
   END_IF;
   IF "step_1" THEN "step_43" := FALSE; END_IF;
END_REGION

REGION Network 33: Unloading procedure first step
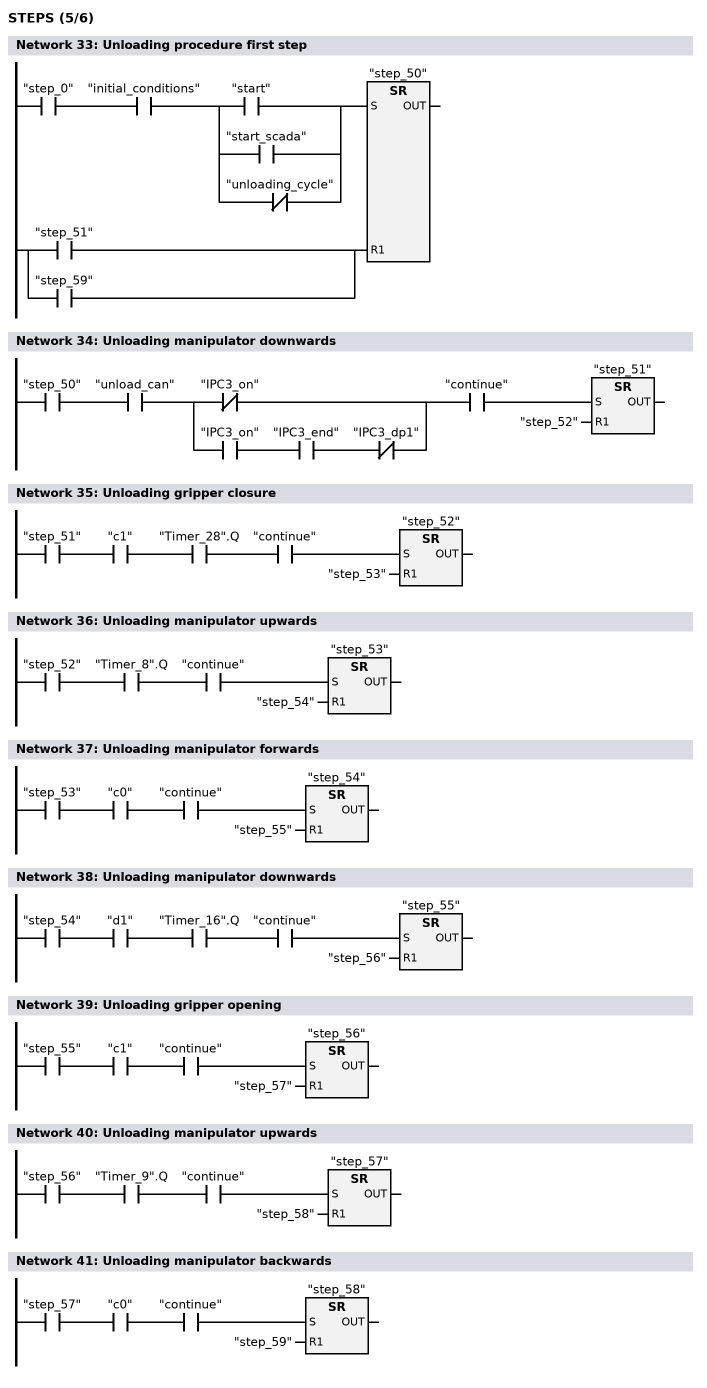
   RUNG wire#powerrail
      Contact( "step_0" )
      Contact( "initial_conditions" )
      wire#w1
      Contact( "start" )
      wire#w2
      S_SR(operand := "step_50", r1 := wire#w3)
   END_RUNG
   RUNG wire#w1
      Contact( "start_scada" )
   END_RUNG wire#w2
   RUNG wire#w1
      I_Contact( "unloading_cycle" )
   END_RUNG wire#w2
   RUNG wire#powerrail
      Contact( "step_51" )
   END_RUNG wire#w3
   RUNG wire#powerrail
      Contact( "step_59" )
   END_RUNG wire#w3
   // the same network as SCL:
   IF "step_0" AND "initial_conditions" AND ("start" OR "start_scada" OR NOT "unloading_cycle") THEN
       "step_50" := TRUE;   // SR flip-flop
   END_IF;
   IF "step_51" OR "step_59" THEN "step_50" := FALSE; END_IF;
END_REGION

REGION Network 34: Unloading manipulator downwards
   RUNG wire#powerrail
      Contact( "step_50" )
      Contact( "unload_can" )
      wire#w1
      I_Contact( "IPC3_on" )
      wire#w2
      Contact( "continue" )
      S_SR(operand := "step_51", r1 := "step_52")
   END_RUNG
   RUNG wire#w1
      Contact( "IPC3_on" )
      Contact( "IPC3_end" )
      I_Contact( "IPC3_dp1" )
   END_RUNG wire#w2
   // the same network as SCL:
   IF "step_50" AND "unload_can" AND (NOT "IPC3_on" OR ("IPC3_on" AND "IPC3_end" AND NOT "IPC3_dp1")) AND "continue" THEN
       "step_51" := TRUE;   // SR flip-flop
   END_IF;
   IF "step_52" THEN "step_51" := FALSE; END_IF;
END_REGION

REGION Network 35: Unloading gripper closure
   RUNG wire#powerrail
      Contact( "step_51" )
      Contact( "c1" )
      Contact( "Timer_28".Q )
      Contact( "continue" )
      S_SR(operand := "step_52", r1 := "step_53")
   END_RUNG
   // the same network as SCL:
   IF "step_51" AND "c1" AND "Timer_28".Q AND "continue" THEN
       "step_52" := TRUE;   // SR flip-flop
   END_IF;
   IF "step_53" THEN "step_52" := FALSE; END_IF;
END_REGION

REGION Network 36: Unloading manipulator upwards
   RUNG wire#powerrail
      Contact( "step_52" )
      Contact( "Timer_8".Q )
      Contact( "continue" )
      S_SR(operand := "step_53", r1 := "step_54")
   END_RUNG
   // the same network as SCL:
   IF "step_52" AND "Timer_8".Q AND "continue" THEN
       "step_53" := TRUE;   // SR flip-flop
   END_IF;
   IF "step_54" THEN "step_53" := FALSE; END_IF;
END_REGION

REGION Network 37: Unloading manipulator forwards
   RUNG wire#powerrail
      Contact( "step_53" )
      Contact( "c0" )
      Contact( "continue" )
      S_SR(operand := "step_54", r1 := "step_55")
   END_RUNG
   // the same network as SCL:
   IF "step_53" AND "c0" AND "continue" THEN
       "step_54" := TRUE;   // SR flip-flop
   END_IF;
   IF "step_55" THEN "step_54" := FALSE; END_IF;
END_REGION

REGION Network 38: Unloading manipulator downwards
   RUNG wire#powerrail
      Contact( "step_54" )
      Contact( "d1" )
      Contact( "Timer_16".Q )
      Contact( "continue" )
      S_SR(operand := "step_55", r1 := "step_56")
   END_RUNG
   // the same network as SCL:
   IF "step_54" AND "d1" AND "Timer_16".Q AND "continue" THEN
       "step_55" := TRUE;   // SR flip-flop
   END_IF;
   IF "step_56" THEN "step_55" := FALSE; END_IF;
END_REGION

REGION Network 39: Unloading gripper opening
   RUNG wire#powerrail
      Contact( "step_55" )
      Contact( "c1" )
      Contact( "continue" )
      S_SR(operand := "step_56", r1 := "step_57")
   END_RUNG
   // the same network as SCL:
   IF "step_55" AND "c1" AND "continue" THEN
       "step_56" := TRUE;   // SR flip-flop
   END_IF;
   IF "step_57" THEN "step_56" := FALSE; END_IF;
END_REGION

REGION Network 40: Unloading manipulator upwards
   RUNG wire#powerrail
      Contact( "step_56" )
      Contact( "Timer_9".Q )
      Contact( "continue" )
      S_SR(operand := "step_57", r1 := "step_58")
   END_RUNG
   // the same network as SCL:
   IF "step_56" AND "Timer_9".Q AND "continue" THEN
       "step_57" := TRUE;   // SR flip-flop
   END_IF;
   IF "step_58" THEN "step_57" := FALSE; END_IF;
END_REGION

REGION Network 41: Unloading manipulator backwards
   RUNG wire#powerrail
      Contact( "step_57" )
      Contact( "c0" )
      Contact( "continue" )
      S_SR(operand := "step_58", r1 := "step_59")
   END_RUNG
   // the same network as SCL:
   IF "step_57" AND "c0" AND "continue" THEN
       "step_58" := TRUE;   // SR flip-flop
   END_IF;
   IF "step_59" THEN "step_58" := FALSE; END_IF;
END_REGION

REGION Network 42: Unloading procedure last step
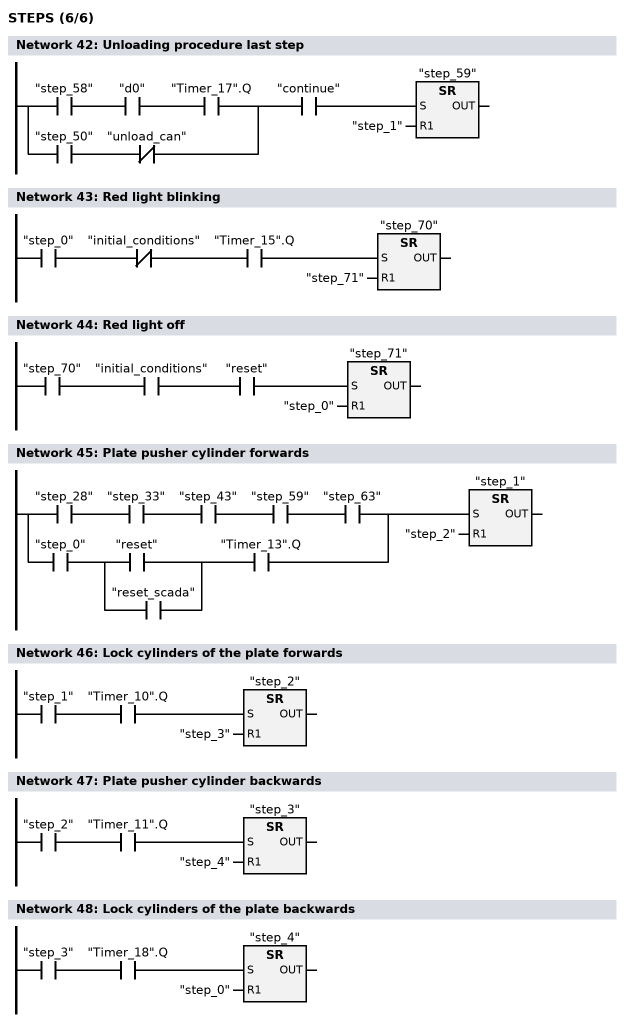
   RUNG wire#powerrail
      Contact( "step_58" )
      Contact( "d0" )
      Contact( "Timer_17".Q )
      wire#w1
      Contact( "continue" )
      S_SR(operand := "step_59", r1 := "step_1")
   END_RUNG
   RUNG wire#powerrail
      Contact( "step_50" )
      I_Contact( "unload_can" )
   END_RUNG wire#w1
   // the same network as SCL:
   IF (("step_58" AND "d0" AND "Timer_17".Q) OR ("step_50" AND NOT "unload_can")) AND "continue" THEN
       "step_59" := TRUE;   // SR flip-flop
   END_IF;
   IF "step_1" THEN "step_59" := FALSE; END_IF;
END_REGION

REGION Network 43: Red light blinking
   RUNG wire#powerrail
      Contact( "step_0" )
      I_Contact( "initial_conditions" )
      Contact( "Timer_15".Q )
      S_SR(operand := "step_70", r1 := "step_71")
   END_RUNG
   // the same network as SCL:
   IF "step_0" AND NOT "initial_conditions" AND "Timer_15".Q THEN
       "step_70" := TRUE;   // SR flip-flop
   END_IF;
   IF "step_71" THEN "step_70" := FALSE; END_IF;
END_REGION

REGION Network 44: Red light off
   RUNG wire#powerrail
      Contact( "step_70" )
      Contact( "initial_conditions" )
      Contact( "reset" )
      S_SR(operand := "step_71", r1 := "step_0")
   END_RUNG
   // the same network as SCL:
   IF "step_70" AND "initial_conditions" AND "reset" THEN
       "step_71" := TRUE;   // SR flip-flop
   END_IF;
   IF "step_0" THEN "step_71" := FALSE; END_IF;
END_REGION

REGION Network 45: Plate pusher cylinder forwards
   RUNG wire#powerrail
      Contact( "step_28" )
      Contact( "step_33" )
      Contact( "step_43" )
      Contact( "step_59" )
      Contact( "step_63" )
      wire#w1
      S_SR(operand := "step_1", r1 := "step_2")
   END_RUNG
   RUNG wire#powerrail
      Contact( "step_0" )
      wire#w2
      Contact( "reset" )
      wire#w3
      Contact( "Timer_13".Q )
   END_RUNG wire#w1
   RUNG wire#w2
      Contact( "reset_scada" )
   END_RUNG wire#w3
   // the same network as SCL:
   IF ("step_28" AND "step_33" AND "step_43" AND "step_59" AND "step_63") OR ("step_0" AND ("reset" OR "reset_scada") AND "Timer_13".Q) THEN
       "step_1" := TRUE;   // SR flip-flop
   END_IF;
   IF "step_2" THEN "step_1" := FALSE; END_IF;
END_REGION

REGION Network 46: Lock cylinders of the plate forwards
   RUNG wire#powerrail
      Contact( "step_1" )
      Contact( "Timer_10".Q )
      S_SR(operand := "step_2", r1 := "step_3")
   END_RUNG
   // the same network as SCL:
   IF "step_1" AND "Timer_10".Q THEN
       "step_2" := TRUE;   // SR flip-flop
   END_IF;
   IF "step_3" THEN "step_2" := FALSE; END_IF;
END_REGION

REGION Network 47: Plate pusher cylinder backwards
   RUNG wire#powerrail
      Contact( "step_2" )
      Contact( "Timer_11".Q )
      S_SR(operand := "step_3", r1 := "step_4")
   END_RUNG
   // the same network as SCL:
   IF "step_2" AND "Timer_11".Q THEN
       "step_3" := TRUE;   // SR flip-flop
   END_IF;
   IF "step_4" THEN "step_3" := FALSE; END_IF;
END_REGION

REGION Network 48: Lock cylinders of the plate backwards
   RUNG wire#powerrail
      Contact( "step_3" )
      Contact( "Timer_18".Q )
      S_SR(operand := "step_4", r1 := "step_0")
   END_RUNG
   // the same network as SCL:
   IF "step_3" AND "Timer_18".Q THEN
       "step_4" := TRUE;   // SR flip-flop
   END_IF;
   IF "step_0" THEN "step_4" := FALSE; END_IF;
END_REGION
END_FUNCTION

FUNCTION "WORKBITS" : Void   // FC2, LAD
TITLE = WORKBITS
{ S7_Optimized_Access := 'TRUE' }
VERSION : 0.1
   VAR_TEMP   // added for the SCL form of the ladder/FBD networks
      _w1 : Bool;
   END_VAR
BEGIN

REGION Network 1: Continue program secuence
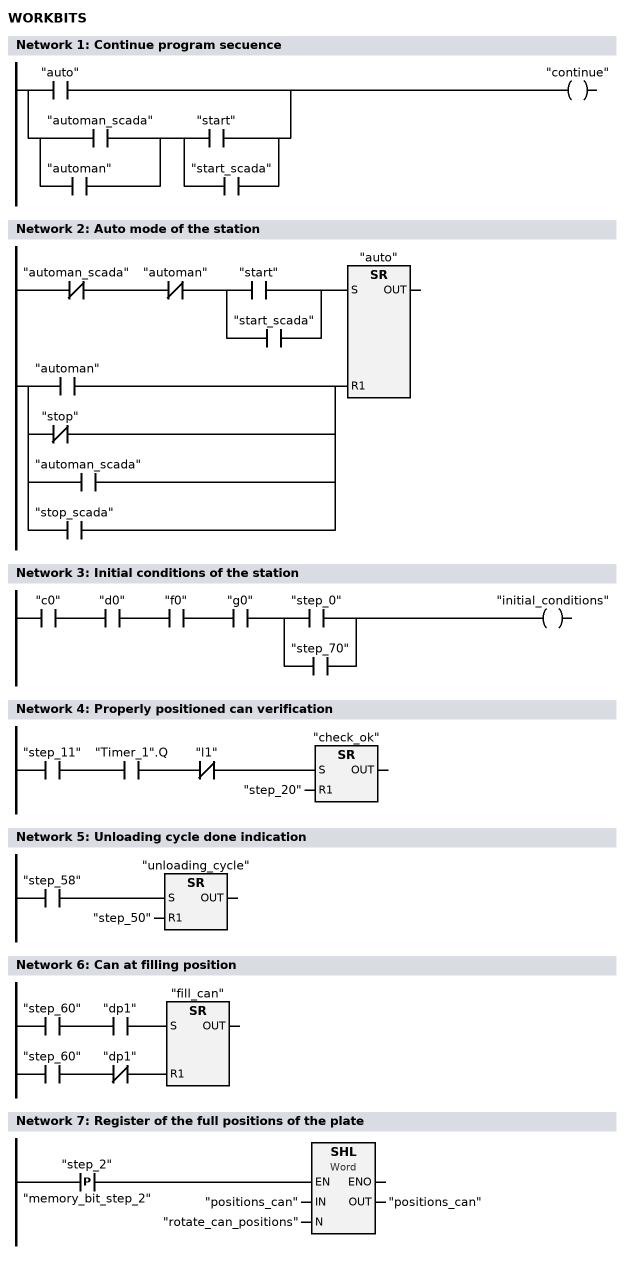
   RUNG wire#powerrail
      Contact( "auto" )
      wire#w1
      Coil( "continue" )
   END_RUNG
   RUNG wire#powerrail
      Contact( "automan_scada" )
      wire#w2
      Contact( "start" )
   END_RUNG wire#w1
   RUNG wire#powerrail
      Contact( "automan" )
   END_RUNG wire#w2
   RUNG wire#w2
      Contact( "start_scada" )
   END_RUNG wire#w1
   // the same network as SCL:
   "continue" := "auto" OR (("automan_scada" OR "automan") AND ("start" OR "start_scada"));
END_REGION

REGION Network 2: Auto mode of the station
   RUNG wire#powerrail
      I_Contact( "automan_scada" )
      I_Contact( "automan" )
      wire#w1
      Contact( "start" )
      wire#w2
      S_SR(operand := "auto", r1 := wire#w3)
   END_RUNG
   RUNG wire#w1
      Contact( "start_scada" )
   END_RUNG wire#w2
   RUNG wire#powerrail
      Contact( "automan" )
   END_RUNG wire#w3
   RUNG wire#powerrail
      I_Contact( "stop" )
   END_RUNG wire#w3
   RUNG wire#powerrail
      Contact( "automan_scada" )
   END_RUNG wire#w3
   RUNG wire#powerrail
      Contact( "stop_scada" )
   END_RUNG wire#w3
   // the same network as SCL:
   IF NOT "automan_scada" AND NOT "automan" AND ("start" OR "start_scada") THEN
       "auto" := TRUE;   // SR flip-flop
   END_IF;
   IF "automan" OR NOT "stop" OR "automan_scada" OR "stop_scada" THEN "auto" := FALSE; END_IF;
END_REGION

REGION Network 3: Initial conditions of the station
   RUNG wire#powerrail
      Contact( "c0" )
      Contact( "d0" )
      Contact( "f0" )
      Contact( "g0" )
      wire#w1
      Contact( "step_0" )
      wire#w2
      Coil( "initial_conditions" )
   END_RUNG
   RUNG wire#w1
      Contact( "step_70" )
   END_RUNG wire#w2
   // the same network as SCL:
   "initial_conditions" := "c0" AND "d0" AND "f0" AND "g0" AND ("step_0" OR "step_70");
END_REGION

REGION Network 4: Properly positioned can verification
   RUNG wire#powerrail
      Contact( "step_11" )
      Contact( "Timer_1".Q )
      I_Contact( "l1" )
      S_SR(operand := "check_ok", r1 := "step_20")
   END_RUNG
   // the same network as SCL:
   IF "step_11" AND "Timer_1".Q AND NOT "l1" THEN
       "check_ok" := TRUE;   // SR flip-flop
   END_IF;
   IF "step_20" THEN "check_ok" := FALSE; END_IF;
END_REGION

REGION Network 5: Unloading cycle done indication
   RUNG wire#powerrail
      Contact( "step_58" )
      S_SR(operand := "unloading_cycle", r1 := "step_50")
   END_RUNG
   // the same network as SCL:
   IF "step_58" THEN
       "unloading_cycle" := TRUE;   // SR flip-flop
   END_IF;
   IF "step_50" THEN "unloading_cycle" := FALSE; END_IF;
END_REGION

REGION Network 6: Can at filling position
   RUNG wire#powerrail
      Contact( "step_60" )
      Contact( "dp1" )
      S_SR(operand := "fill_can", r1 := wire#w1)
   END_RUNG
   RUNG wire#powerrail
      Contact( "step_60" )
      I_Contact( "dp1" )
   END_RUNG wire#w1
   // the same network as SCL:
   IF "step_60" AND "dp1" THEN
       "fill_can" := TRUE;   // SR flip-flop
   END_IF;
   IF "step_60" AND NOT "dp1" THEN "fill_can" := FALSE; END_IF;
END_REGION

REGION Network 7: Register of the full positions of the plate
   RUNG wire#powerrail
      P_Contact(operand := "step_2", bit := "memory_bit_step_2")
      { S7_Templates := "SrcType := Word"; S7_GenerateENO := "TRUE" } Shl(in := "positions_can", n := "rotate_can_positions", out => "positions_can")
   END_RUNG
   // the same network as SCL:
   #_w1 := "step_2" AND NOT "memory_bit_step_2";   // rising edge of "step_2"
   "memory_bit_step_2" := "step_2";
   IF #_w1 THEN "positions_can" := SHL(IN := "positions_can", N := "rotate_can_positions"); END_IF;
END_REGION
END_FUNCTION

FUNCTION "TIMERS" : Void   // FC3, LAD
TITLE = TIMERS
{ S7_Optimized_Access := 'TRUE' }
VERSION : 0.1
BEGIN

REGION Network 1: Timer 0
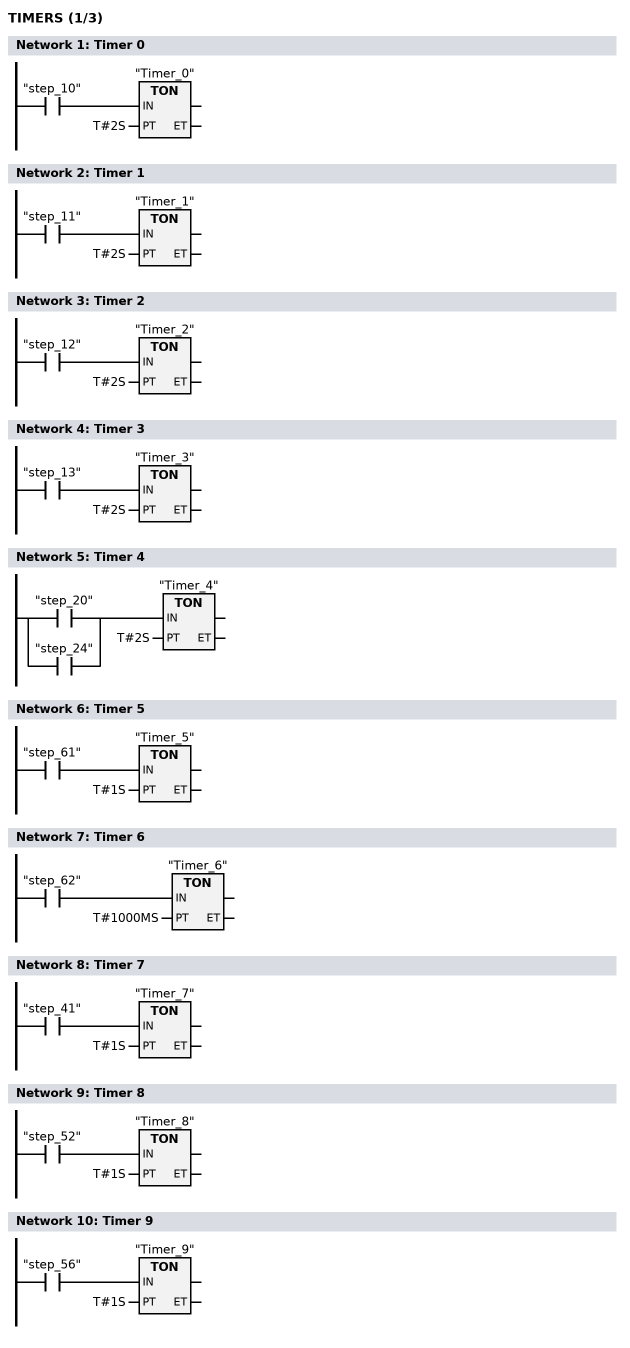
   "Timer_0".TON(IN := "step_10", PT := T#2S);
END_REGION

REGION Network 2: Timer 1
   "Timer_1".TON(IN := "step_11", PT := T#2S);
END_REGION

REGION Network 3: Timer 2
   "Timer_2".TON(IN := "step_12", PT := T#2S);
END_REGION

REGION Network 4: Timer 3
   "Timer_3".TON(IN := "step_13", PT := T#2S);
END_REGION

REGION Network 5: Timer 4
   "Timer_4".TON(IN := "step_20" OR "step_24", PT := T#2S);
END_REGION

REGION Network 6: Timer 5
   "Timer_5".TON(IN := "step_61", PT := T#1S);
END_REGION

REGION Network 7: Timer 6
   "Timer_6".TON(IN := "step_62", PT := T#1000MS);
END_REGION

REGION Network 8: Timer 7
   "Timer_7".TON(IN := "step_41", PT := T#1S);
END_REGION

REGION Network 9: Timer 8
   "Timer_8".TON(IN := "step_52", PT := T#1S);
END_REGION

REGION Network 10: Timer 9
   "Timer_9".TON(IN := "step_56", PT := T#1S);
END_REGION

REGION Network 11: Timer 10
